KUKA KRL program: MyProgram_154().src

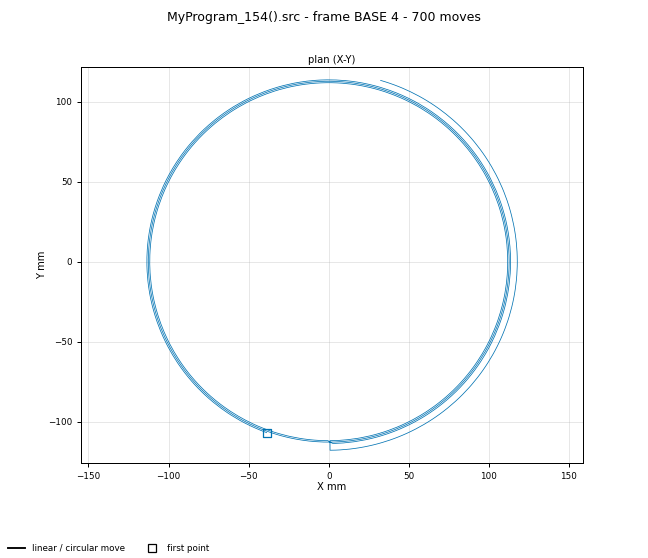
[picture p0: tool path of MyProgram_154().src in frame BASE 4, 700 of 700 moves have a stored position in this frame; points joined in program order, loops and branches not executed]
&ACCESS RVP
&REL 1
&PARAM TEMPLATE = C:\KRC\Roboter\Template\vorgabe
&PARAM EDITMASK = *
DEF MyProgram_154()
; ---- Setting reference (Base) ----
$BASE = BASE_DATA[4]

; --------------------------
; ---- Setting tool (TCP) ----
$TOOL = TOOL_DATA[3]
; --------------------------

$VEL.CP = VEL_APROX_PRINT
Startdeposition()
$VEL.CP = VEL_PRINT
LIN {X -38.7795,Y -106.7145,Z 119,A -114.0854,B 24.9553,C -1.5455,E1 24.9444,E2 200.0846} C_DIS
LIN {X -42.2899,Y -105.3741,Z 119,A -116.1743,B 24.9556,C -1.5393,E1 24.9389,E2 202.1927} C_DIS
LIN {X -46.3885,Y -103.634,Z 119,A -118.1057,B 24.9547,C -1.5549,E1 24.9341,E2 204.0916} C_DIS
LIN {X -48.9846,Y -102.4323,Z 119,A -120.2238,B 24.9562,C -1.5287,E1 24.9286,E2 206.2774} C_DIS
LIN {X -52.6968,Y -100.573,Z 119,A -121.7129,B 24.9546,C -1.5564,E1 24.925,E2 207.7047} C_DIS
LIN {X -55.5486,Y -99.0263,Z 119,A -123.3546,B 24.9545,C -1.5584,E1 24.921,E2 209.3463} C_DIS
LIN {X -60.9242,Y -95.8139,Z 119,A -126.6405,B 24.9545,C -1.5579,E1 24.9132,E2 212.6435} C_DIS
LIN {X -63.1418,Y -94.368,Z 119,A -128.2578,B 24.9551,C -1.5485,E1 24.9093,E2 214.2885} C_DIS
LIN {X -67.1706,Y -91.542,Z 119,A -130.4641,B 24.9542,C -1.5641,E1 24.9044,E2 216.4654} C_DIS
LIN {X -70.0841,Y -89.3319,Z 119,A -132.2235,B 24.9538,C -1.571,E1 24.9005,E2 218.2149} C_DIS
LIN {X -71.9862,Y -87.8078,Z 119,A -133.5514,B 24.9538,C -1.5692,E1 24.8976,E2 219.5519} C_DIS
LIN {X -74.7924,Y -85.428,Z 119,A -135.353,B 24.9535,C -1.5751,E1 24.8938,E2 221.3466} C_DIS
LIN {X -77.6668,Y -82.8234,Z 119,A -137.329,B 24.9533,C -1.5784,E1 24.8898,E2 223.3229} C_DIS
LIN {X -81.3821,Y -79.1774,Z 119,A -140.0426,B 24.9532,C -1.5804,E1 24.8844,E2 226.043} C_DIS
LIN {X -83.7193,Y -76.7001,Z 119,A -141.611,B 24.9526,C -1.5904,E1 24.8814,E2 227.5946} C_DIS
LIN {X -85.8302,Y -74.3318,Z 119,A -143.3683,B 24.9528,C -1.5877,E1 24.8782,E2 229.3661} C_DIS
LIN {X -88.2166,Y -71.4818,Z 119,A -145.143,B 24.9523,C -1.5962,E1 24.875,E2 231.1288} C_DIS
LIN {X -90.1414,Y -69.0395,Z 119,A -147.103,B 24.953,C -1.5844,E1 24.8716,E2 233.1262} C_DIS
LIN {X -92.0799,Y -66.4339,Z 119,A -148.4579,B 24.952,C -1.5998,E1 24.8694,E2 234.451} C_DIS
LIN {X -94.3065,Y -63.2327,Z 119,A -151.3484,B 24.9539,C -1.5684,E1 24.8648,E2 237.4308} C_DIS
LIN {X -97.447,Y -58.2773,Z 119,A -153.2453,B 24.9509,C -1.6182,E1 24.8622,E2 239.2187} C_DIS
LIN {X -100.3495,Y -53.1211,Z 119,A -156.2923,B 24.9506,C -1.6239,E1 24.8581,E2 242.2681} C_DIS
LIN {X -101.8163,Y -50.2524,Z 119,A -157.9977,B 24.9505,C -1.6253,E1 24.8559,E2 243.9793} C_DIS
LIN {X -103.469,Y -46.7547,Z 119,A -160.1125,B 24.9505,C -1.6245,E1 24.8534,E2 246.1077} C_DIS
LIN {X -105.0495,Y -43.0873,Z 119,A -161.9877,B 24.9499,C -1.6359,E1 24.8514,E2 247.9662} C_DIS
LIN {X -107.1276,Y -37.6231,Z 119,A -164.846,B 24.9491,C -1.6482,E1 24.8486,E2 250.811} C_DIS
LIN {X -108.4347,Y -33.6711,Z 119,A -167.0827,B 24.9491,C -1.6492,E1 24.8467,E2 253.0583} C_DIS
LIN {X -109.4832,Y -30.0915,Z 119,A -169.0013,B 24.9488,C -1.6535,E1 24.8452,E2 254.9776} C_DIS
LIN {X -110.3079,Y -26.9068,Z 119,A -170.6364,B 24.9484,C -1.6597,E1 24.8441,E2 256.6076} C_DIS
LIN {X -111.1636,Y -23.1205,Z 119,A -172.5881,B 24.948,C -1.6661,E1 24.8429,E2 258.5555} C_DIS
LIN {X -111.7921,Y -19.8596,Z 119,A -174.5884,B 24.9484,C -1.6587,E1 24.8419,E2 260.5853} C_DIS
LIN {X -112.5109,Y -15.2835,Z 119,A -176.6425,B 24.9473,C -1.6772,E1 24.8411,E2 262.6076} C_DIS
LIN {X -112.9126,Y -11.9401,Z 119,A -178.5887,B 24.9475,C -1.673,E1 24.8405,E2 264.5754} C_DIS
LIN {X -113.3804,Y -6.0614,Z 119,A 178.5739,B 24.9466,C -1.688,E1 24.84,E2 267.3941} C_DIS
LIN {X -113.5197,Y -2.2658,Z 119,A 176.7243,B 24.946,C -1.6968,E1 24.8398,E2 269.2338} C_DIS
LIN {X -113.5092,Y 2.8146,Z 119,A 173.8444,B 24.9463,C -1.6928,E1 24.8398,E2 272.1406} C_DIS
LIN {X -113.2912,Y 7.5449,Z 119,A 171.7176,B 24.9451,C -1.7109,E1 24.8402,E2 274.2372} C_DIS
LIN {X -113.0207,Y 10.8788,Z 119,A 170.163,B 24.9445,C -1.7216,E1 24.8406,E2 275.7756} C_DIS
LIN {X -112.6461,Y 14.2411,Z 119,A 168.2727,B 24.9445,C -1.72,E1 24.8412,E2 277.6811} C_DIS
LIN {X -112.0315,Y 18.4615,Z 119,A 166.1494,B 24.944,C -1.7281,E1 24.8421,E2 279.7977} C_DIS
LIN {X -111.4363,Y 21.7683,Z 119,A 164.3501,B 24.944,C -1.7295,E1 24.843,E2 281.6042} C_DIS
LIN {X -110.5057,Y 26.0885,Z 119,A 161.6768,B 24.9446,C -1.7195,E1 24.8447,E2 284.3172} C_DIS
LIN {X -109.5791,Y 29.7363,Z 119,A 160.2216,B 24.9431,C -1.7428,E1 24.8457,E2 285.7252} C_DIS
LIN {X -108.4418,Y 33.648,Z 119,A 157.5317,B 24.9443,C -1.7247,E1 24.848,E2 288.4737} C_DIS
LIN {X -106.9969,Y 37.9954,Z 119,A 155.7728,B 24.9424,C -1.7533,E1 24.8496,E2 290.1743} C_DIS
LIN {X -105.7047,Y 41.4529,Z 119,A 154.0435,B 24.9417,C -1.7644,E1 24.8513,E2 291.8871} C_DIS
LIN {X -103.2381,Y 47.267,Z 119,A 150.8158,B 24.9411,C -1.7725,E1 24.8548,E2 295.1133} C_DIS
LIN {X -101.4731,Y 50.9447,Z 119,A 148.6316,B 24.9411,C -1.7737,E1 24.8575,E2 297.3062} C_DIS
LIN {X -99.5576,Y 54.5927,Z 119,A 146.5283,B 24.9407,C -1.779,E1 24.8603,E2 299.4083} C_DIS
LIN {X -97.1628,Y 58.7474,Z 119,A 144.0709,B 24.9403,C -1.7845,E1 24.8638,E2 301.8651} C_DIS
LIN {X -95.0134,Y 62.1645,Z 119,A 142.116,B 24.9397,C -1.7935,E1 24.8667,E2 303.8084} C_DIS
LIN {X -91.9767,Y 66.5766,Z 119,A 139.0093,B 24.9403,C -1.7852,E1 24.8717,E2 306.9502} C_DIS
LIN {X -89.9849,Y 69.2426,Z 119,A 137.365,B 24.9399,C -1.7911,E1 24.8745,E2 308.5882} C_DIS
LIN {X -87.9451,Y 71.8168,Z 119,A 136.1646,B 24.9384,C -1.8135,E1 24.8766,E2 309.7409} C_DIS
LIN {X -85.2574,Y 74.9865,Z 119,A 133.7554,B 24.9388,C -1.8066,E1 24.881,E2 312.1775} C_DIS
LIN {X -80.3903,Y 80.1843,Z 119,A 130.2401,B 24.938,C -1.8186,E1 24.8878,E2 315.6795} C_DIS
LIN {X -77.9973,Y 82.5126,Z 119,A 128.0362,B 24.9391,C -1.8021,E1 24.8923,E2 317.9316} C_DIS
LIN {X -74.8259,Y 85.3987,Z 119,A 125.7336,B 24.9391,C -1.8016,E1 24.8972,E2 320.2445} C_DIS
LIN {X -71.0662,Y 88.5534,Z 119,A 123.8711,B 24.9371,C -1.8314,E1 24.9011,E2 322.0433} C_DIS
LIN {X -68.7439,Y 90.3689,Z 119,A 121.8998,B 24.9382,C -1.8153,E1 24.9056,E2 324.0599} C_DIS
LIN {X -65.3509,Y 92.8521,Z 119,A 120.2399,B 24.9367,C -1.838,E1 24.9092,E2 325.6716} C_DIS
LIN {X -61.8864,Y 95.1962,Z 119,A 118.1045,B 24.9365,C -1.8411,E1 24.9142,E2 327.8066} C_DIS
LIN {X -59.1389,Y 96.925,Z 119,A 115.4465,B 24.939,C -1.8036,E1 24.9208,E2 330.562} C_DIS
LIN {X -53.3558,Y 100.2259,Z 119,A 113.1232,B 24.9358,C -1.8507,E1 24.9262,E2 332.7797} C_DIS
LIN {X -50.2914,Y 101.7969,Z 119,A 111.6116,B 24.935,C -1.8628,E1 24.9299,E2 334.2669} C_DIS
LIN {X -46.3293,Y 103.6607,Z 119,A 109.3479,B 24.9349,C -1.8639,E1 24.9357,E2 336.5333} C_DIS
LIN {X -40.3596,Y 106.127,Z 119,A 105.8317,B 24.9353,C -1.858,E1 24.9448,E2 340.0714} C_DIS
LIN {X -36.0067,Y 107.682,Z 119,A 103.3217,B 24.9356,C -1.8537,E1 24.9515,E2 342.5964} C_DIS
LIN {X -31.3299,Y 109.1348,Z 119,A 101.1768,B 24.9345,C -1.8698,E1 24.9571,E2 344.7067} C_DIS
LIN {X -28.2896,Y 109.9614,Z 119,A 99.6621,B 24.9341,C -1.8745,E1 24.9612,E2 346.2124} C_DIS
LIN {X -22.2676,Y 111.3387,Z 119,A 96.426,B 24.9343,C -1.8724,E1 24.9701,E2 349.4577} C_DIS
LIN {X -18.8866,Y 111.9604,Z 119,A 94.8799,B 24.9336,C -1.8815,E1 24.9742,E2 350.9837} C_DIS
LIN {X -13.7991,Y 112.7021,Z 119,A 92.1188,B 24.934,C -1.8762,E1 24.9819,E2 353.7596} C_DIS
LIN {X -7.9378,Y 113.2647,Z 119,A 89.1949,B 24.9338,C -1.8797,E1 24.99,E2 356.6768} C_DIS
LIN {X -5.1434,Y 113.4259,Z 119,A 87.1623,B 24.9355,C -1.8543,E1 24.9959,E2 358.77} C_DIS
LIN {X -1.0062,Y 113.5381,Z 119,A 85.4495,B 24.9344,C -1.8704,E1 25.0006,E2 360.4446} C_DIS
LIN {X 4.6202,Y 113.4484,Z 119,A 82.9834,B 24.9333,C -1.8865,E1 25.0073,E2 362.8722} C_DIS
LIN {X 10.4517,Y 113.0601,Z 119,A 79.3073,B 24.9354,C -1.8557,E1 25.0178,E2 366.6194} C_DIS
LIN {X 14.4604,Y 112.6176,Z 119,A 77.7972,B 24.9339,C -1.8775,E1 25.0218,E2 368.0768} C_DIS
LIN {X 17.49,Y 112.1871,Z 119,A 75.8625,B 24.9351,C -1.8604,E1 25.0272,E2 370.0501} C_DIS
LIN {X 20.9601,Y 111.5919,Z 119,A 74.3788,B 24.9343,C -1.8721,E1 25.0312,E2 371.5044} C_DIS
LIN {X 25.1759,Y 110.7165,Z 119,A 72.3191,B 24.934,C -1.8759,E1 25.0368,E2 373.5525} C_DIS
LIN {X 28.519,Y 109.9025,Z 119,A 70.6003,B 24.934,C -1.8756,E1 25.0415,E2 375.2693} C_DIS
LIN {X 32.1679,Y 108.8901,Z 119,A 68.6954,B 24.9341,C -1.8745,E1 25.0466,E2 377.1736} C_DIS
LIN {X 35.545,Y 107.8367,Z 119,A 66.9758,B 24.9341,C -1.8759,E1 25.0511,E2 378.8868} C_DIS
LIN {X 37.8064,Y 107.0633,Z 119,A 65.6314,B 24.9345,C -1.8689,E1 25.0547,E2 380.2451} C_DIS
LIN {X 42.254,Y 105.3886,Z 119,A 63.2762,B 24.9345,C -1.8684,E1 25.0609,E2 382.5965} C_DIS
LIN {X 45.7399,Y 103.9223,Z 119,A 60.8053,B 24.9364,C -1.8419,E1 25.0673,E2 385.1239} C_DIS
LIN {X 49.6347,Y 102.1199,Z 119,A 59.1837,B 24.935,C -1.8628,E1 25.0713,E2 386.6919} C_DIS
LIN {X 53.4516,Y 100.1754,Z 119,A 56.6902,B 24.9362,C -1.8455,E1 25.0775,E2 389.2194} C_DIS
LIN {X 56.3394,Y 98.5787,Z 119,A 55.1408,B 24.936,C -1.8481,E1 25.0813,E2 390.7579} C_DIS
LIN {X 60.8663,Y 95.851,Z 119,A 52.6168,B 24.9358,C -1.8503,E1 25.0872,E2 393.2688} C_DIS
LIN {X 64.1193,Y 93.7061,Z 119,A 50.6128,B 24.9362,C -1.8454,E1 25.0919,E2 395.2776} C_DIS
LIN {X 67.6543,Y 91.1875,Z 119,A 48.5006,B 24.9362,C -1.845,E1 25.0966,E2 397.3834} C_DIS
LIN {X 71.9271,Y 87.8557,Z 119,A 45.7992,B 24.9364,C -1.8413,E1 25.1025,E2 400.0833} C_DIS
LIN {X 74.6558,Y 85.5473,Z 119,A 44.2974,B 24.9358,C -1.8512,E1 25.1057,E2 401.5558} C_DIS
LIN {X 78.3837,Y 82.1471,Z 119,A 41.4962,B 24.9369,C -1.8346,E1 25.1115,E2 404.3849} C_DIS
LIN {X 81.1101,Y 79.4556,Z 119,A 39.7544,B 24.9366,C -1.839,E1 25.1149,E2 406.109} C_DIS
LIN {X 84.2332,Y 76.1372,Z 119,A 37.2848,B 24.9375,C -1.8262,E1 25.1196,E2 408.598} C_DIS
LIN {X 86.7497,Y 73.2567,Z 119,A 34.8821,B 24.9392,C -1.8005,E1 25.124,E2 411.0503} C_DIS
LIN {X 89.3227,Y 70.0958,Z 119,A 33.3055,B 24.9381,C -1.817,E1 25.1267,E2 412.5805} C_DIS
LIN {X 91.5873,Y 67.1087,Z 119,A 31.7955,B 24.9373,C -1.8296,E1 25.1292,E2 414.0537} C_DIS
LIN {X 93.2489,Y 64.78,Z 119,A 30.0633,B 24.9384,C -1.8128,E1 25.132,E2 415.8169} C_DIS
LIN {X 94.9753,Y 62.2223,Z 119,A 28.4277,B 24.9389,C -1.8052,E1 25.1345,E2 417.4624} C_DIS
LIN {X 96.9762,Y 59.0546,Z 119,A 26.5962,B 24.9391,C -1.8029,E1 25.1372,E2 419.2901} C_DIS
LIN {X 98.9328,Y 55.7161,Z 119,A 24.6472,B 24.9394,C -1.7977,E1 25.1399,E2 421.2412} C_DIS
LIN {X 100.7803,Y 52.303,Z 119,A 22.8234,B 24.9394,C -1.7984,E1 25.1423,E2 423.0538} C_DIS
LIN {X 104.3637,Y 44.7269,Z 119,A 18.6192,B 24.9401,C -1.7874,E1 25.1473,E2 427.2613} C_DIS
LIN {X 106.2287,Y 40.0912,Z 119,A 16.0223,B 24.9408,C -1.7765,E1 25.15,E2 429.8695} C_DIS
LIN {X 107.5213,Y 36.4834,Z 119,A 14.1733,B 24.941,C -1.7746,E1 25.1517,E2 431.7127} C_DIS
LIN {X 108.4396,Y 33.6552,Z 119,A 12.6614,B 24.9413,C -1.7695,E1 25.1529,E2 433.228} C_DIS
LIN {X 109.6687,Y 29.4048,Z 119,A 10.3479,B 24.942,C -1.7589,E1 25.1547,E2 435.5532} C_DIS
LIN {X 110.5233,Y 26.0121,Z 119,A 8.1985,B 24.9435,C -1.7358,E1 25.1561,E2 437.7445} C_DIS
LIN {X 111.3121,Y 22.397,Z 119,A 6.9312,B 24.9421,C -1.7574,E1 25.1568,E2 438.9535} C_DIS
LIN {X 112.0752,Y 18.197,Z 119,A 4.421,B 24.9436,C -1.7342,E1 25.158,E2 441.5036} C_DIS
LIN {X 112.6423,Y 14.2702,Z 119,A 1.9254,B 24.9455,C -1.7053,E1 25.1589,E2 444.0527} C_DIS
LIN {X 113.1592,Y 9.3219,Z 119,A -0.513,B 24.9458,C -1.7005,E1 25.1595,E2 446.4881} C_DIS
LIN {X 113.4497,Y 4.59,Z 119,A -2.2614,B 24.9444,C -1.7222,E1 25.1597,E2 448.1749} C_DIS
LIN {X 113.5358,Y 1.3367,Z 119,A -3.9301,B 24.9448,C -1.7156,E1 25.1597,E2 449.8491} C_DIS
LIN {X 113.5269,Y -1.8736,Z 119,A -5.7164,B 24.9457,C -1.7027,E1 25.1597,E2 451.6552} C_DIS
LIN {X 113.3099,Y -7.2693,Z 119,A -7.9332,B 24.9447,C -1.7173,E1 25.1594,E2 453.8247} C_DIS
LIN {X 112.6463,Y -14.239,Z 119,A -11.8061,B 24.9465,C -1.69,E1 25.1583,E2 457.7389} C_DIS
LIN {X 111.7509,Y -20.0885,Z 119,A -14.4516,B 24.9461,C -1.696,E1 25.1572,E2 460.3546} C_DIS
LIN {X 110.4229,Y -26.4358,Z 119,A -17.8457,B 24.9471,C -1.6797,E1 25.1552,E2 463.7673} C_DIS
LIN {X 109.6822,Y -29.3549,Z 119,A -19.3799,B 24.9475,C -1.6742,E1 25.1541,E2 465.3058} C_DIS
LIN {X 108.6814,Y -32.8714,Z 119,A -21.317,B 24.9481,C -1.6641,E1 25.1525,E2 467.2557} C_DIS
LIN {X 107.5918,Y -36.2743,Z 119,A -22.9036,B 24.9478,C -1.6684,E1 25.1512,E2 468.8232} C_DIS
LIN {X 106.354,Y -39.7601,Z 119,A -24.9096,B 24.9486,C -1.6561,E1 25.1493,E2 470.8469} C_DIS
LIN {X 103.6092,Y -46.4435,Z 119,A -28.1919,B 24.9483,C -1.6616,E1 25.1458,E2 474.0982} C_DIS
LIN {X 101.598,Y -50.6927,Z 119,A -30.8862,B 24.9496,C -1.6395,E1 25.1425,E2 476.83} C_DIS
LIN {X 99.7763,Y -54.1897,Z 119,A -33.2879,B 24.9511,C -1.6147,E1 25.1392,E2 479.2775} C_DIS
LIN {X 97.8977,Y -57.5148,Z 119,A -34.6108,B 24.9498,C -1.6367,E1 25.1375,E2 480.5418} C_DIS
LIN {X 94.8546,Y -62.4054,Z 119,A -37.612,B 24.9506,C -1.624,E1 25.133,E2 483.5578} C_DIS
LIN {X 93.2011,Y -64.8488,Z 119,A -38.953,B 24.9504,C -1.6266,E1 25.1309,E2 484.8861} C_DIS
LIN {X 91.3605,Y -67.4186,Z 119,A -40.6904,B 24.9511,C -1.6156,E1 25.128,E2 486.641} C_DIS
LIN {X 89.2292,Y -70.2141,Z 119,A -42.384,B 24.9511,C -1.6145,E1 25.1251,E2 488.3292} C_DIS
LIN {X 87.0673,Y -72.8784,Z 119,A -44.2734,B 24.9519,C -1.6027,E1 25.1217,E2 490.2378} C_DIS
LIN {X 84.57,Y -75.7611,Z 119,A -46.063,B 24.9519,C -1.6038,E1 25.1184,E2 492.0166} C_DIS
LIN {X 81.984,Y -78.5529,Z 119,A -48.0162,B 24.9522,C -1.5975,E1 25.1147,E2 493.9763} C_DIS
LIN {X 79.4027,Y -81.1624,Z 119,A -49.9139,B 24.9526,C -1.5908,E1 25.1109,E2 495.8816} C_DIS
LIN {X 76.7767,Y -83.649,Z 119,A -51.633,B 24.9526,C -1.5913,E1 25.1074,E2 497.5926} C_DIS
LIN {X 73.944,Y -86.1642,Z 119,A -53.5598,B 24.9529,C -1.5862,E1 25.1034,E2 499.5239} C_DIS
LIN {X 71.6521,Y -88.0786,Z 119,A -55.058,B 24.953,C -1.5832,E1 25.1001,E2 501.0235} C_DIS
LIN {X 68.6736,Y -90.4218,Z 119,A -57.0278,B 24.9534,C -1.5764,E1 25.0958,E2 503.002} C_DIS
LIN {X 66.0008,Y -92.3889,Z 119,A -58.6322,B 24.9534,C -1.5761,E1 25.0921,E2 504.6015} C_DIS
LIN {X 62.724,Y -94.6446,Z 119,A -60.4684,B 24.9532,C -1.5798,E1 25.0879,E2 506.4229} C_DIS
LIN {X 60.2833,Y -96.2173,Z 119,A -62.0206,B 24.9536,C -1.573,E1 25.0843,E2 507.9861} C_DIS
LIN {X 57.7569,Y -97.7546,Z 119,A -63.5157,B 24.9538,C -1.5701,E1 25.0807,E2 509.4834} C_DIS
LIN {X 53.4628,Y -100.1696,Z 119,A -66.1549,B 24.9545,C -1.5588,E1 25.0742,E2 512.1417} C_DIS
LIN {X 50.0811,Y -101.9012,Z 119,A -67.9524,B 24.9543,C -1.5609,E1 25.0697,E2 513.9291} C_DIS
LIN {X 44.5083,Y -104.4551,Z 119,A -71.2636,B 24.9552,C -1.5465,E1 25.0612,E2 517.2663} C_DIS
LIN {X 40.6633,Y -106.012,Z 119,A -73.3415,B 24.9553,C -1.5442,E1 25.0558,E2 519.345} C_DIS
LIN {X 36.415,Y -107.5443,Z 119,A -75.407,B 24.9549,C -1.5507,E1 25.0504,E2 521.3909} C_DIS
LIN {X 33.2505,Y -108.5651,Z 119,A -77.1473,B 24.9552,C -1.546,E1 25.0458,E2 523.1393} C_DIS
LIN {X 30.1039,Y -109.4798,Z 119,A -78.6676,B 24.955,C -1.55,E1 25.0417,E2 524.6476} C_DIS
LIN {X 26.8253,Y -110.3278,Z 119,A -80.324,B 24.955,C -1.5506,E1 25.0372,E2 526.3002} C_DIS
LIN {X 22.8635,Y -111.2164,Z 119,A -82.5574,B 24.9555,C -1.5406,E1 25.0311,E2 528.5543} C_DIS
LIN {X 15.9868,Y -112.411,Z 119,A -86.1378,B 24.9558,C -1.5354,E1 25.0212,E2 532.1434} C_DIS
LIN {X 9.0633,Y -113.1798,Z 119,A -90.5647,B 24.9582,C -1.4943,E1 25.0086,E2 536.6649} C_DIS
LIN {X 2.6596,Y -113.5124,Z 119,A -93.7317,B 24.9581,C -1.4962,E1 24.9998,E2 539.8268} C_DIS
LIN {X 2.6596,Y -113.5124,Z 119,A -93.7317,B 24.9581,C -1.4962,E1 24.9998,E2 539.8268} C_DIS
Enddeposition()
LIN {X 0.7947,Y -112.634,Z 119,A -93.4663,B 24.9542,C -1.5636,E1 25.001,E2 539.4018} C_DIS
Startdeposition()
$VEL.CP = VEL_PRINT
LIN {X 3.6315,Y -112.5922,Z 119,A -91.4349,B 24.9527,C -1.5892,E1 25.0068,E2 537.3099} C_DIS
LIN {X 9.3853,Y -112.2597,Z 119,A -88.603,B 24.9529,C -1.5862,E1 25.0147,E2 534.4866} C_DIS
LIN {X 14.6247,Y -111.6973,Z 119,A -85.9699,B 24.9529,C -1.5857,E1 25.022,E2 531.8565} C_DIS
LIN {X 17.4837,Y -111.2859,Z 119,A -84.4862,B 24.9528,C -1.5874,E1 25.0261,E2 530.3701} C_DIS
LIN {X 20.076,Y -110.8473,Z 119,A -82.5788,B 24.9512,C -1.6137,E1 25.0315,E2 528.4026} C_DIS
LIN {X 23.8423,Y -110.0987,Z 119,A -81.0612,B 24.9523,C -1.5961,E1 25.0355,E2 526.9285} C_DIS
LIN {X 27.3941,Y -109.271,Z 119,A -79.1677,B 24.9521,C -1.5996,E1 25.0407,E2 525.0295} C_DIS
LIN {X 31.0805,Y -108.2788,Z 119,A -77.4071,B 24.9524,C -1.5937,E1 25.0454,E2 523.2856} C_DIS
LIN {X 34.4302,Y -107.2604,Z 119,A -75.5291,B 24.952,C -1.6002,E1 25.0504,E2 521.3958} C_DIS
LIN {X 37.9515,Y -106.0675,Z 119,A -73.1772,B 24.9506,C -1.6232,E1 25.0567,E2 518.9941} C_DIS
LIN {X 41.4531,Y -104.7467,Z 119,A -71.8213,B 24.9519,C -1.6014,E1 25.0601,E2 517.6929} C_DIS
LIN {X 47.4616,Y -102.1644,Z 119,A -68.809,B 24.9525,C -1.5923,E1 25.0678,E2 514.7093} C_DIS
LIN {X 50.1295,Y -100.8821,Z 119,A -66.9839,B 24.9515,C -1.6091,E1 25.0724,E2 512.8494} C_DIS
LIN {X 53.2616,Y -99.2654,Z 119,A -65.1317,B 24.9511,C -1.6148,E1 25.077,E2 510.9888} C_DIS
LIN {X 57.1934,Y -97.052,Z 119,A -62.9315,B 24.9511,C -1.6148,E1 25.0823,E2 508.7954} C_DIS
LIN {X 59.8016,Y -95.467,Z 119,A -61.1759,B 24.9504,C -1.6269,E1 25.0866,E2 507.0167} C_DIS
LIN {X 63.4757,Y -93.0652,Z 119,A -59.1345,B 24.9507,C -1.6227,E1 25.0913,E2 504.992} C_DIS
LIN {X 66.5163,Y -90.9161,Z 119,A -57.2466,B 24.9504,C -1.6264,E1 25.0955,E2 503.102} C_DIS
LIN {X 69.2022,Y -88.8905,Z 119,A -55.4209,B 24.9499,C -1.6353,E1 25.0996,E2 501.262} C_DIS
LIN {X 72.0223,Y -86.6195,Z 119,A -53.6859,B 24.9499,C -1.6346,E1 25.1033,E2 499.5353} C_DIS
LIN {X 74.8907,Y -84.1526,Z 119,A -51.7388,B 24.9496,C -1.6401,E1 25.1074,E2 497.583} C_DIS
LIN {X 77.4696,Y -81.7849,Z 119,A -49.9042,B 24.9492,C -1.6468,E1 25.1112,E2 495.7399} C_DIS
LIN {X 80.1076,Y -79.2019,Z 119,A -48.1676,B 24.9492,C -1.6449,E1 25.1146,E2 494.0151} C_DIS
LIN {X 82.5016,Y -76.7076,Z 119,A -46.3106,B 24.9487,C -1.6539,E1 25.1182,E2 492.145} C_DIS
LIN {X 84.8864,Y -74.0571,Z 119,A -44.5965,B 24.9487,C -1.654,E1 25.1214,E2 490.4382} C_DIS
LIN {X 87.368,Y -71.1129,Z 119,A -42.6253,B 24.9484,C -1.6598,E1 25.1249,E2 488.4624} C_DIS
LIN {X 89.4115,Y -68.5261,Z 119,A -41.0209,B 24.9483,C -1.661,E1 25.1276,E2 486.8628} C_DIS
LIN {X 91.5304,Y -65.6691,Z 119,A -38.8766,B 24.947,C -1.6815,E1 25.1312,E2 484.6805} C_DIS
LIN {X 93.5113,Y -62.8169,Z 119,A -37.2723,B 24.9472,C -1.679,E1 25.1337,E2 483.0901} C_DIS
LIN {X 97.5682,Y -56.3084,Z 119,A -33.5204,B 24.9469,C -1.6833,E1 25.1391,E2 479.347} C_DIS
LIN {X 99.4537,Y -52.9087,Z 119,A -31.5202,B 24.9465,C -1.6903,E1 25.1418,E2 477.3409} C_DIS
LIN {X 101.2342,Y -49.4193,Z 119,A -29.415,B 24.9457,C -1.7015,E1 25.1444,E2 475.2206} C_DIS
LIN {X 102.9456,Y -45.7461,Z 119,A -27.4796,B 24.9457,C -1.702,E1 25.1467,E2 473.2946} C_DIS
LIN {X 105.0232,Y -40.7492,Z 119,A -24.6819,B 24.945,C -1.7126,E1 25.1496,E2 470.4872} C_DIS
LIN {X 106.3578,Y -37.1242,Z 119,A -22.9296,B 24.9453,C -1.7089,E1 25.1512,E2 468.7534} C_DIS
LIN {X 107.4241,Y -33.9199,Z 119,A -21.0792,B 24.9445,C -1.7205,E1 25.1528,E2 466.8862} C_DIS
LIN {X 108.4494,Y -30.4786,Z 119,A -19.2611,B 24.9442,C -1.726,E1 25.1543,E2 465.0656} C_DIS
LIN {X 109.5508,Y -26.2486,Z 119,A -17.2319,B 24.9442,C -1.7241,E1 25.1556,E2 463.0526} C_DIS
LIN {X 110.4204,Y -22.3072,Z 119,A -15.1724,B 24.9438,C -1.731,E1 25.1568,E2 460.9887} C_DIS
LIN {X 111.0009,Y -19.2193,Z 119,A -13.4091,B 24.943,C -1.7439,E1 25.1577,E2 459.2055} C_DIS
LIN {X 111.7852,Y -13.9466,Z 119,A -10.8296,B 24.9428,C -1.7466,E1 25.1587,E2 456.6347} C_DIS
LIN {X 112.3337,Y -8.4596,Z 119,A -8.174,B 24.9427,C -1.7488,E1 25.1594,E2 453.9897} C_DIS
LIN {X 112.5698,Y -4.2983,Z 119,A -5.6678,B 24.941,C -1.7736,E1 25.1597,E2 451.4398} C_DIS
LIN {X 112.6514,Y -0.0991,Z 119,A -3.5805,B 24.9407,C -1.7783,E1 25.1597,E2 449.3538} C_DIS
LIN {X 112.5859,Y 3.8355,Z 119,A -0.8985,B 24.9381,C -1.8167,E1 25.1595,E2 446.5974} C_DIS
LIN {X 112.2447,Y 9.5723,Z 119,A 1.1622,B 24.9402,C -1.7857,E1 25.1591,E2 444.6219} C_DIS
LIN {X 111.6524,Y 14.9717,Z 119,A 3.7608,B 24.9402,C -1.787,E1 25.1582,E2 442.0357} C_DIS
LIN {X 110.6446,Y 21.1646,Z 119,A 6.6735,B 24.9403,C -1.7842,E1 25.1569,E2 439.1465} C_DIS
LIN {X 109.7837,Y 25.2527,Z 119,A 9.1378,B 24.9388,C -1.8065,E1 25.1554,E2 436.6439} C_DIS
LIN {X 108.999,Y 28.4524,Z 119,A 10.6712,B 24.9389,C -1.8052,E1 25.1544,E2 435.1227} C_DIS
LIN {X 108.1951,Y 31.376,Z 119,A 12.3655,B 24.9381,C -1.8169,E1 25.1531,E2 433.4104} C_DIS
LIN {X 107.1483,Y 34.7766,Z 119,A 14.1339,B 24.9379,C -1.8205,E1 25.1516,E2 431.6435} C_DIS
LIN {X 105.8415,Y 38.5711,Z 119,A 16.1402,B 24.9376,C -1.825,E1 25.1497,E2 429.6378} C_DIS
LIN {X 104.2185,Y 42.764,Z 119,A 18.34,B 24.9374,C -1.8278,E1 25.1475,E2 427.4437} C_DIS
LIN {X 103.0183,Y 45.5824,Z 119,A 20.0598,B 24.9366,C -1.8397,E1 25.1455,E2 425.7052} C_DIS
LIN {X 100.3962,Y 51.0959,Z 119,A 22.739,B 24.9373,C -1.829,E1 25.1424,E2 423.0656} C_DIS
LIN {X 98.553,Y 54.5676,Z 119,A 25.0731,B 24.9359,C -1.8498,E1 25.1392,E2 420.6946} C_DIS
LIN {X 96.685,Y 57.8143,Z 119,A 26.852,B 24.9359,C -1.8492,E1 25.1367,E2 418.9263} C_DIS
LIN {X 94.8595,Y 60.7605,Z 119,A 28.6349,B 24.9355,C -1.8548,E1 25.134,E2 417.1393} C_DIS
LIN {X 93.0192,Y 63.5437,Z 119,A 30.2592,B 24.9355,C -1.8559,E1 25.1315,E2 415.5205} C_DIS
LIN {X 91.6445,Y 65.5092,Z 119,A 31.5461,B 24.935,C -1.862,E1 25.1294,E2 414.2254} C_DIS
LIN {X 89.559,Y 68.3347,Z 119,A 33.4497,B 24.9343,C -1.8718,E1 25.1262,E2 412.3078} C_DIS
LIN {X 86.938,Y 71.639,Z 119,A 35.5237,B 24.9342,C -1.8737,E1 25.1226,E2 410.239} C_DIS
LIN {X 84.814,Y 74.14,Z 119,A 37.1383,B 24.9341,C -1.8751,E1 25.1196,E2 408.6282} C_DIS
LIN {X 82.4097,Y 76.8052,Z 119,A 39.1339,B 24.9333,C -1.8869,E1 25.1158,E2 406.6136} C_DIS
LIN {X 79.115,Y 80.1933,Z 119,A 41.359,B 24.9335,C -1.8841,E1 25.1115,E2 404.4046} C_DIS
LIN {X 75.6509,Y 83.4719,Z 119,A 43.8839,B 24.9328,C -1.8935,E1 25.1063,E2 401.8678} C_DIS
LIN {X 72.9859,Y 85.8092,Z 119,A 45.5649,B 24.9329,C -1.8916,E1 25.1028,E2 400.1978} C_DIS
LIN {X 70.1723,Y 88.1258,Z 119,A 47.5785,B 24.9322,C -1.9023,E1 25.0984,E2 398.1667} C_DIS
LIN {X 66.7518,Y 90.7437,Z 119,A 49.5934,B 24.9324,C -1.8984,E1 25.0939,E2 396.1683} C_DIS
LIN {X 63.6728,Y 92.9318,Z 119,A 51.4063,B 24.9326,C -1.8968,E1 25.0898,E2 394.3653} C_DIS
LIN {X 61.1664,Y 94.599,Z 119,A 53.1385,B 24.9317,C -1.9082,E1 25.0857,E2 392.6119} C_DIS
LIN {X 58.6522,Y 96.1774,Z 119,A 55.7458,B 24.928,C -1.9595,E1 25.0792,E2 389.8912} C_DIS
LIN {X 52.6274,Y 99.6019,Z 119,A 57.8893,B 24.9321,C -1.9029,E1 25.0743,E2 387.8879} C_DIS
LIN {X 50.0218,Y 100.9355,Z 119,A 59.5599,B 24.9314,C -1.9128,E1 25.07,E2 386.1984} C_DIS
LIN {X 46.1351,Y 102.7703,Z 119,A 61.6921,B 24.9314,C -1.913,E1 25.0646,E2 384.0712} C_DIS
LIN {X 43.4758,Y 103.9235,Z 119,A 63.3061,B 24.9308,C -1.9207,E1 25.0605,E2 382.4427} C_DIS
LIN {X 39.2626,Y 105.5891,Z 119,A 65.4173,B 24.9313,C -1.9145,E1 25.055,E2 380.3507} C_DIS
LIN {X 35.7967,Y 106.8119,Z 119,A 66.9886,B 24.9321,C -1.9033,E1 25.051,E2 378.8093} C_DIS
LIN {X 33.5511,Y 107.5384,Z 119,A 68.5603,B 24.9309,C -1.9203,E1 25.0467,E2 377.2002} C_DIS
LIN {X 30.061,Y 108.5677,Z 119,A 70.3307,B 24.931,C -1.9181,E1 25.0419,E2 375.438} C_DIS
LIN {X 27.8574,Y 109.152,Z 119,A 71.5005,B 24.931,C -1.9193,E1 25.0388,E2 374.2671} C_DIS
LIN {X 24.4877,Y 109.9579,Z 119,A 73.3366,B 24.9306,C -1.9234,E1 25.0337,E2 372.4238} C_DIS
LIN {X 21.3615,Y 110.6067,Z 119,A 74.863,B 24.9309,C -1.92,E1 25.0296,E2 370.9074} C_DIS
LIN {X 18.29,Y 111.1563,Z 119,A 76.4751,B 24.9308,C -1.9216,E1 25.0252,E2 369.2931} C_DIS
LIN {X 15.6813,Y 111.5539,Z 119,A 77.8491,B 24.9306,C -1.9233,E1 25.0213,E2 367.9163} C_DIS
LIN {X 12.539,Y 111.952,Z 119,A 79.5061,B 24.9305,C -1.9256,E1 25.0167,E2 366.2551} C_DIS
LIN {X 8.6877,Y 112.3155,Z 119,A 81.624,B 24.93,C -1.9322,E1 25.0108,E2 364.1228} C_DIS
LIN {X 4.7207,Y 112.5517,Z 119,A 83.5167,B 24.9304,C -1.9266,E1 25.0056,E2 362.2439} C_DIS
LIN {X 0.6724,Y 112.6486,Z 119,A 85.8653,B 24.9295,C -1.9386,E1 24.9989,E2 359.8671} C_DIS
LIN {X -2.5326,Y 112.623,Z 119,A 87.2746,B 24.9303,C -1.9288,E1 24.9951,E2 358.481} C_DIS
LIN {X -5.8185,Y 112.5009,Z 119,A 88.9345,B 24.9303,C -1.9277,E1 24.9904,E2 356.8234} C_DIS
LIN {X -9.8873,Y 112.2168,Z 119,A 91.0695,B 24.9303,C -1.9293,E1 24.9845,E2 354.6836} C_DIS
LIN {X -13.2277,Y 111.8713,Z 119,A 92.6185,B 24.9308,C -1.9217,E1 24.9802,E2 353.1517} C_DIS
LIN {X -17.2817,Y 111.3171,Z 119,A 94.3792,B 24.9318,C -1.9069,E1 24.9755,E2 351.4246} C_DIS
LIN {X -19.4135,Y 110.9664,Z 119,A 95.9601,B 24.9304,C -1.9262,E1 24.971,E2 349.7965} C_DIS
LIN {X -22.8708,Y 110.3047,Z 119,A 97.5601,B 24.9311,C -1.9168,E1 24.9667,E2 348.2169} C_DIS
LIN {X -27.0893,Y 109.3457,Z 119,A 99.7345,B 24.9313,C -1.9136,E1 24.9608,E2 346.0471} C_DIS
LIN {X -30.2716,Y 108.508,Z 119,A 101.5936,B 24.9309,C -1.9196,E1 24.9557,E2 344.171} C_DIS
LIN {X -34.149,Y 107.351,Z 119,A 103.9729,B 24.9301,C -1.9305,E1 24.9493,E2 341.7615} C_DIS
LIN {X -37.4393,Y 106.2472,Z 119,A 105.2703,B 24.9317,C -1.909,E1 24.946,E2 340.5128} C_DIS
LIN {X -40.2691,Y 105.2079,Z 119,A 107.7177,B 24.9291,C -1.9447,E1 24.9394,E2 337.9753} C_DIS
LIN {X -45.2689,Y 103.155,Z 119,A 109.6447,B 24.9318,C -1.9067,E1 24.9347,E2 336.1342} C_DIS
LIN {X -48.7254,Y 101.5677,Z 119,A 111.5159,B 24.9322,C -1.9011,E1 24.9299,E2 334.2715} C_DIS
LIN {X -51.7702,Y 100.0516,Z 119,A 113.3893,B 24.932,C -1.9041,E1 24.9252,E2 332.386} C_DIS
LIN {X -56.7579,Y 97.3094,Z 119,A 116.1061,B 24.9329,C -1.8917,E1 24.9187,E2 329.6907} C_DIS
LIN {X -59.9092,Y 95.3997,Z 119,A 118.0575,B 24.9329,C -1.8914,E1 24.914,E2 327.7341} C_DIS
LIN {X -63.2264,Y 93.234,Z 119,A 120.1046,B 24.9331,C -1.8887,E1 24.9093,E2 325.6865} C_DIS
LIN {X -66.4102,Y 90.9938,Z 119,A 122.39,B 24.9325,C -1.897,E1 24.904,E2 323.3735} C_DIS
LIN {X -69.7329,Y 88.4731,Z 119,A 124.6587,B 24.9325,C -1.8984,E1 24.899,E2 321.0931} C_DIS
LIN {X -72.4847,Y 86.2324,Z 119,A 126.2201,B 24.9334,C -1.8845,E1 24.8957,E2 319.5588} C_DIS
LIN {X -76.1549,Y 83.0095,Z 119,A 128.8601,B 24.9334,C -1.885,E1 24.8902,E2 316.907} C_DIS
LIN {X -79.2536,Y 80.0564,Z 119,A 131.6627,B 24.932,C -1.905,E1 24.8846,E2 314.045} C_DIS
LIN {X -83.2506,Y 75.8922,Z 119,A 133.8808,B 24.9345,C -1.8686,E1 24.8805,E2 311.9037} C_DIS
LIN {X -86.6876,Y 71.9404,Z 119,A 136.2597,B 24.9358,C -1.8504,E1 24.8762,E2 309.5576} C_DIS
LIN {X -88.6176,Y 69.5501,Z 119,A 138.7621,B 24.9335,C -1.8837,E1 24.8718,E2 306.9638} C_DIS
LIN {X -91.779,Y 65.3207,Z 119,A 140.62,B 24.9363,C -1.8432,E1 24.8689,E2 305.1934} C_DIS
LIN {X -93.2639,Y 63.1822,Z 119,A 141.9935,B 24.9364,C -1.8415,E1 24.8667,E2 303.8172} C_DIS
LIN {X -95.4963,Y 59.7547,Z 119,A 144.0525,B 24.9369,C -1.8347,E1 24.8636,E2 301.7639} C_DIS
LIN {X -97.6107,Y 56.2345,Z 119,A 146.8566,B 24.9354,C -1.8571,E1 24.8596,E2 298.8919} C_DIS
LIN {X -99.9054,Y 52.051,Z 119,A 148.5338,B 24.9379,C -1.8201,E1 24.8575,E2 297.294} C_DIS
LIN {X -101.5371,Y 48.7891,Z 119,A 150.4776,B 24.938,C -1.818,E1 24.8551,E2 295.3447} C_DIS
LIN {X -103.3382,Y 44.8486,Z 119,A 152.6665,B 24.9385,C -1.8107,E1 24.8526,E2 293.1612} C_DIS
LIN {X -104.8606,Y 41.1633,Z 119,A 154.7017,B 24.9389,C -1.8048,E1 24.8505,E2 291.1289} C_DIS
LIN {X -106.1927,Y 37.5948,Z 119,A 156.778,B 24.9389,C -1.8042,E1 24.8485,E2 289.0422} C_DIS
LIN {X -107.7489,Y 32.8724,Z 119,A 159.3249,B 24.9395,C -1.7969,E1 24.8463,E2 286.4981} C_DIS
LIN {X -108.7761,Y 29.2905,Z 119,A 161.1838,B 24.94,C -1.7894,E1 24.845,E2 284.6462} C_DIS
LIN {X -109.5649,Y 26.1908,Z 119,A 162.8452,B 24.9402,C -1.7856,E1 24.8439,E2 282.9843} C_DIS
LIN {X -110.2992,Y 22.8976,Z 119,A 164.5513,B 24.9406,C -1.7796,E1 24.8429,E2 281.2822} C_DIS
LIN {X -110.9418,Y 19.5504,Z 119,A 166.2997,B 24.941,C -1.7746,E1 24.842,E2 279.5355} C_DIS
LIN {X -111.4852,Y 16.165,Z 119,A 167.8086,B 24.942,C -1.7598,E1 24.8414,E2 278.053} C_DIS
LIN {X -111.7832,Y 13.9619,Z 119,A 169.0572,B 24.9419,C -1.7607,E1 24.8409,E2 276.7948} C_DIS
LIN {X -112.0526,Y 11.5929,Z 119,A 170.3541,B 24.9419,C -1.7601,E1 24.8405,E2 275.4915} C_DIS
LIN {X -112.3463,Y 8.3024,Z 119,A 172.1499,B 24.942,C -1.7591,E1 24.8401,E2 273.6873} C_DIS
LIN {X -112.5521,Y 4.7119,Z 119,A 173.8932,B 24.9426,C -1.7498,E1 24.8399,E2 271.9557} C_DIS
LIN {X -112.6444,Y 1.3551,Z 119,A 175.7384,B 24.9426,C -1.7496,E1 24.8398,E2 270.0998} C_DIS
LIN {X -112.6188,Y -2.7636,Z 119,A 177.7952,B 24.9432,C -1.7413,E1 24.8398,E2 268.0503} C_DIS
LIN {X -112.4574,Y -6.6052,Z 119,A 179.5646,B 24.9441,C -1.7277,E1 24.8401,E2 266.3028} C_DIS
LIN {X -112.2401,Y -9.6269,Z 119,A -178.841,B 24.9442,C -1.7248,E1 24.8405,E2 264.7057} C_DIS
LIN {X -111.9575,Y -12.4922,Z 119,A -177.3715,B 24.9445,C -1.7203,E1 24.8409,E2 263.2381} C_DIS
LIN {X -111.5173,Y -15.9393,Z 119,A -175.445,B 24.9445,C -1.721,E1 24.8416,E2 261.2986} C_DIS
LIN {X -110.9805,Y -19.3356,Z 119,A -173.8519,B 24.9452,C -1.7093,E1 24.8423,E2 259.7239} C_DIS
LIN {X -110.4669,Y -22.0809,Z 119,A -172.1982,B 24.9449,C -1.714,E1 24.8432,E2 258.0491} C_DIS
LIN {X -109.6155,Y -25.9811,Z 119,A -170.3333,B 24.9458,C -1.7011,E1 24.8444,E2 256.204} C_DIS
LIN {X -108.7764,Y -29.2892,Z 119,A -168.5543,B 24.946,C -1.6975,E1 24.8456,E2 254.4233} C_DIS
LIN {X -107.8023,Y -32.7001,Z 119,A -166.4608,B 24.9456,C -1.7034,E1 24.8473,E2 252.3035} C_DIS
LIN {X -106.5438,Y -36.5921,Z 119,A -164.5851,B 24.9465,C -1.689,E1 24.849,E2 250.4514} C_DIS
LIN {X -104.9578,Y -40.9156,Z 119,A -162.3281,B 24.9472,C -1.6787,E1 24.8512,E2 248.2063} C_DIS
LIN {X -103.7339,Y -43.9256,Z 119,A -160.5009,B 24.9471,C -1.6808,E1 24.8531,E2 246.3639} C_DIS
LIN {X -102.172,Y -47.4452,Z 119,A -158.6464,B 24.9477,C -1.6711,E1 24.8553,E2 244.5225} C_DIS
LIN {X -100.7425,Y -50.411,Z 119,A -156.9907,B 24.948,C -1.6656,E1 24.8573,E2 242.871} C_DIS
LIN {X -99.4866,Y -52.8463,Z 119,A -155.2553,B 24.9474,C -1.6754,E1 24.8596,E2 241.1029} C_DIS
LIN {X -96.9948,Y -57.2901,Z 119,A -152.9209,B 24.9485,C -1.6581,E1 24.8628,E2 238.7976} C_DIS
LIN {X -94.9948,Y -60.5497,Z 119,A -150.6118,B 24.9479,C -1.6676,E1 24.8663,E2 236.4542} C_DIS
LIN {X -92.3744,Y -64.4761,Z 119,A -148.5759,B 24.9492,C -1.6467,E1 24.8694,E2 234.4579} C_DIS
LIN {X -90.3518,Y -67.2825,Z 119,A -146.9607,B 24.9498,C -1.6365,E1 24.8721,E2 232.8592} C_DIS
LIN {X -88.72,Y -69.4205,Z 119,A -145.3534,B 24.9494,C -1.6428,E1 24.8749,E2 231.2291} C_DIS
LIN {X -86.5606,Y -72.0932,Z 119,A -143.6114,B 24.9497,C -1.6385,E1 24.8779,E2 229.4895} C_DIS
LIN {X -84.0625,Y -74.9913,Z 119,A -141.7081,B 24.9501,C -1.6323,E1 24.8814,E2 227.5923} C_DIS
LIN {X -82.1254,Y -77.1076,Z 119,A -140.2285,B 24.9502,C -1.6298,E1 24.8842,E2 226.112} C_DIS
LIN {X -79.4861,Y -79.8268,Z 119,A -138.2981,B 24.9505,C -1.6258,E1 24.888,E2 224.183} C_DIS
LIN {X -77.1762,Y -82.0609,Z 119,A -136.677,B 24.9507,C -1.6219,E1 24.8913,E2 222.5646} C_DIS
LIN {X -74.7599,Y -84.2696,Z 119,A -134.9575,B 24.9507,C -1.6207,E1 24.8949,E2 220.8409} C_DIS
LIN {X -71.8785,Y -86.739,Z 119,A -133.1099,B 24.9512,C -1.6137,E1 24.8988,E2 219.003} C_DIS
LIN {X -69.252,Y -88.8521,Z 119,A -131.242,B 24.951,C -1.6168,E1 24.9029,E2 217.1208} C_DIS
LIN {X -66.4872,Y -90.9374,Z 119,A -129.5602,B 24.9514,C -1.6104,E1 24.9067,E2 215.4481} C_DIS
LIN {X -62.5397,Y -93.6982,Z 119,A -126.9711,B 24.9514,C -1.6121,E1 24.9127,E2 212.8463} C_DIS
LIN {X -59.6112,Y -95.5859,Z 119,A -124.734,B 24.9503,C -1.6288,E1 24.9181,E2 210.5624} C_DIS
LIN {X -55.9905,Y -97.7509,Z 119,A -123.2723,B 24.9522,C -1.5972,E1 24.9214,E2 209.1716} C_DIS
LIN {X -53.4866,Y -99.1433,Z 119,A -121.67,B 24.952,C -1.6012,E1 24.9254,E2 207.5551} C_DIS
LIN {X -49.443,Y -101.2224,Z 119,A -119.4712,B 24.9524,C -1.5935,E1 24.9308,E2 205.3687} C_DIS
LIN {X -46.0541,Y -102.8068,Z 119,A -117.4324,B 24.9522,C -1.5971,E1 24.9361,E2 203.3165} C_DIS
LIN {X -42.7475,Y -104.2252,Z 119,A -115.6725,B 24.9525,C -1.5922,E1 24.9406,E2 201.5641} C_DIS
LIN {X -38.1197,Y -106.0061,Z 119,A -113.2268,B 24.9528,C -1.5866,E1 24.9469,E2 199.1266} C_DIS
LIN {X -35.5181,Y -106.9059,Z 119,A -111.6052,B 24.9523,C -1.5948,E1 24.9513,E2 197.4824} C_DIS
LIN {X -32.0125,Y -108.0063,Z 119,A -109.8897,B 24.9528,C -1.587,E1 24.9558,E2 195.7826} C_DIS
LIN {X -29.1796,Y -108.806,Z 119,A -108.4063,B 24.9529,C -1.5854,E1 24.9598,E2 194.3006} C_DIS
LIN {X -25.9214,Y -109.6292,Z 119,A -106.7534,B 24.9531,C -1.5821,E1 24.9643,E2 192.6534} C_DIS
LIN {X -22.8984,Y -110.299,Z 119,A -104.9893,B 24.9527,C -1.5894,E1 24.9692,E2 190.8696} C_DIS
LIN {X -19.9769,Y -110.8651,Z 119,A -103.5251,B 24.9528,C -1.5868,E1 24.9732,E2 189.4102} C_DIS
LIN {X -16.5445,Y -111.4311,Z 119,A -101.7311,B 24.9528,C -1.5873,E1 24.9781,E2 187.6133} C_DIS
LIN {X -12.2662,Y -111.982,Z 119,A -99.0779,B 24.9516,C -1.6069,E1 24.9856,E2 184.912} C_DIS
LIN {X -8.4322,Y -112.3359,Z 119,A -97.5262,B 24.9527,C -1.5892,E1 24.9898,E2 183.4016} C_DIS
LIN {X -3.1626,Y -112.6066,Z 119,A -94.936,B 24.9529,C -1.5854,E1 24.997,E2 180.8199} C_DIS
LIN {X 0.7947,Y -112.634,Z 119,A -93.4641,B 24.9542,C -1.5626,E1 25.001,E2 179.4018} C_DIS
Enddeposition()
LIN {X 0.7947,Y -112.634,Z 119,A -93.4641,B 24.9542,C -1.5626,E1 25.001,E2 179.4018} C_DIS
Startdeposition()
$VEL.CP = VEL_PRINT
LIN {X -0.4514,Y -111.7584,Z 119,A -94.2931,B 24.9538,C -1.5698,E1 24.9987,E2 180.2138} C_DIS
LIN {X -2.7919,Y -111.726,Z 119,A -95.4923,B 24.9538,C -1.5696,E1 24.9954,E2 181.4136} C_DIS
LIN {X -5.8749,Y -111.6049,Z 119,A -97.0955,B 24.9538,C -1.5686,E1 24.9909,E2 183.0196} C_DIS
LIN {X -8.8792,Y -111.4057,Z 119,A -98.5573,B 24.9537,C -1.5721,E1 24.9868,E2 184.4738} C_DIS
LIN {X -12.3584,Y -111.0755,Z 119,A -100.4117,B 24.9538,C -1.5696,E1 24.9817,E2 186.3351} C_DIS
LIN {X -15.0639,Y -110.7411,Z 119,A -101.9452,B 24.9542,C -1.5641,E1 24.9774,E2 187.8826} C_DIS
LIN {X -18.1269,Y -110.2796,Z 119,A -103.3253,B 24.9536,C -1.5733,E1 24.9736,E2 189.2422} C_DIS
LIN {X -20.8143,Y -109.8041,Z 119,A -104.6401,B 24.9534,C -1.5773,E1 24.97,E2 190.5488} C_DIS
LIN {X -23.5147,Y -109.2576,Z 119,A -106.2159,B 24.9538,C -1.5711,E1 24.9657,E2 192.1412} C_DIS
LIN {X -25.8351,Y -108.734,Z 119,A -107.5716,B 24.9541,C -1.566,E1 24.962,E2 193.5107} C_DIS
LIN {X -28.8467,Y -107.9724,Z 119,A -109.0317,B 24.9537,C -1.5725,E1 24.958,E2 194.9577} C_DIS
LIN {X -31.1277,Y -107.3388,Z 119,A -110.3833,B 24.954,C -1.5676,E1 24.9544,E2 196.3231} C_DIS
LIN {X -34.1004,Y -106.43,Z 119,A -111.9174,B 24.9537,C -1.5713,E1 24.9503,E2 197.8511} C_DIS
LIN {X -37.0566,Y -105.4367,Z 119,A -113.3717,B 24.9533,C -1.5786,E1 24.9465,E2 199.2909} C_DIS
LIN {X -40.6847,Y -104.0907,Z 119,A -115.3988,B 24.9533,C -1.5786,E1 24.9412,E2 201.322} C_DIS
LIN {X -44.3803,Y -102.5698,Z 119,A -117.4641,B 24.9533,C -1.5801,E1 24.9359,E2 203.3886} C_DIS
LIN {X -46.8766,Y -101.4533,Z 119,A -118.8916,B 24.9532,C -1.5806,E1 24.9322,E2 204.8183} C_DIS
LIN {X -49.4621,Y -100.2178,Z 119,A -120.3293,B 24.953,C -1.5837,E1 24.9286,E2 206.2524} C_DIS
LIN {X -51.8045,Y -99.0276,Z 119,A -121.7163,B 24.953,C -1.5837,E1 24.9252,E2 207.6429} C_DIS
LIN {X -54.2198,Y -97.7261,Z 119,A -123.1422,B 24.953,C -1.5849,E1 24.9217,E2 209.0703} C_DIS
LIN {X -56.6297,Y -96.3495,Z 119,A -124.3831,B 24.9524,C -1.5943,E1 24.9187,E2 210.2924} C_DIS
LIN {X -58.9695,Y -94.9355,Z 119,A -125.9537,B 24.9527,C -1.5896,E1 24.9149,E2 211.8792} C_DIS
LIN {X -61.2559,Y -93.4767,Z 119,A -127.1824,B 24.9521,C -1.5983,E1 24.9121,E2 213.0911} C_DIS
LIN {X -63.2137,Y -92.1659,Z 119,A -128.7057,B 24.9528,C -1.5875,E1 24.9085,E2 214.6451} C_DIS
LIN {X -65.469,Y -90.5779,Z 119,A -130.178,B 24.9528,C -1.5875,E1 24.9052,E2 216.1224} C_DIS
LIN {X -68.2853,Y -88.4715,Z 119,A -131.8642,B 24.9523,C -1.5955,E1 24.9014,E2 217.7959} C_DIS
LIN {X -71.0514,Y -86.2671,Z 119,A -133.72,B 24.9523,C -1.5972,E1 24.8974,E2 219.6546} C_DIS
LIN {X -73.518,Y -84.1735,Z 119,A -135.3217,B 24.9519,C -1.6027,E1 24.894,E2 221.2494} C_DIS
LIN {X -76.0615,Y -81.8852,Z 119,A -137.2158,B 24.9519,C -1.6007,E1 24.8901,E2 223.1561} C_DIS
LIN {X -78.5321,Y -79.516,Z 119,A -138.8468,B 24.9515,C -1.6093,E1 24.8869,E2 224.7733} C_DIS
LIN {X -81.2748,Y -76.7107,Z 119,A -140.8853,B 24.9513,C -1.6126,E1 24.8829,E2 226.8126} C_DIS
LIN {X -83.3959,Y -74.3992,Z 119,A -142.5091,B 24.9511,C -1.6157,E1 24.8799,E2 228.4365} C_DIS
LIN {X -85.8361,Y -71.5701,Z 119,A -144.4191,B 24.9508,C -1.6203,E1 24.8764,E2 230.3441} C_DIS
LIN {X -87.7929,Y -69.1557,Z 119,A -146.0356,B 24.9506,C -1.6232,E1 24.8736,E2 231.9612} C_DIS
LIN {X -90.0171,Y -66.235,Z 119,A -147.6671,B 24.9497,C -1.6377,E1 24.8709,E2 233.566} C_DIS
LIN {X -91.6677,Y -63.9308,Z 119,A -149.2933,B 24.9499,C -1.6346,E1 24.8682,E2 235.2077} C_DIS
LIN {X -93.9971,Y -60.4535,Z 119,A -151.4211,B 24.9495,C -1.6408,E1 24.865,E2 237.3312} C_DIS
LIN {X -95.3449,Y -58.3055,Z 119,A -152.6153,B 24.9491,C -1.6484,E1 24.8632,E2 238.5135} C_DIS
LIN {X -96.556,Y -56.2804,Z 119,A -154.0082,B 24.9493,C -1.6445,E1 24.8612,E2 239.923} C_DIS
LIN {X -97.9759,Y -53.7689,Z 119,A -155.4334,B 24.9489,C -1.6506,E1 24.8593,E2 241.341} C_DIS
LIN {X -99.2038,Y -51.4698,Z 119,A -156.977,B 24.9492,C -1.6462,E1 24.8572,E2 242.9033} C_DIS
LIN {X -100.5659,Y -48.7517,Z 119,A -158.4549,B 24.9487,C -1.6538,E1 24.8554,E2 244.3712} C_DIS
LIN {X -101.7667,Y -46.192,Z 119,A -159.6934,B 24.948,C -1.6661,E1 24.854,E2 245.587} C_DIS
LIN {X -102.867,Y -43.6869,Z 119,A -161.1039,B 24.9477,C -1.6699,E1 24.8524,E2 246.9963} C_DIS
LIN {X -103.9058,Y -41.1554,Z 119,A -162.6992,B 24.948,C -1.6665,E1 24.8507,E2 248.6086} C_DIS
LIN {X -104.7639,Y -38.9237,Z 119,A -164.0563,B 24.948,C -1.665,E1 24.8494,E2 249.9768} C_DIS
LIN {X -105.7995,Y -36.0088,Z 119,A -165.3481,B 24.947,C -1.6812,E1 24.8482,E2 251.2374} C_DIS
LIN {X -106.5366,Y -33.7708,Z 119,A -166.8727,B 24.9476,C -1.6726,E1 24.8469,E2 252.7913} C_DIS
LIN {X -107.7149,Y -29.7998,Z 119,A -168.8728,B 24.9469,C -1.6838,E1 24.8454,E2 254.7762} C_DIS
LIN {X -108.5003,Y -26.7929,Z 119,A -170.303,B 24.9462,C -1.6951,E1 24.8444,E2 256.1879} C_DIS
LIN {X -109.0451,Y -24.4891,Z 119,A -171.8355,B 24.9467,C -1.6865,E1 24.8434,E2 257.7498} C_DIS
LIN {X -109.7,Y -21.355,Z 119,A -173.3929,B 24.9462,C -1.695,E1 24.8426,E2 259.2963} C_DIS
LIN {X -110.3435,Y -17.7441,Z 119,A -175.3809,B 24.946,C -1.6968,E1 24.8416,E2 261.2918} C_DIS
LIN {X -110.7923,Y -14.6709,Z 119,A -176.8481,B 24.9454,C -1.7067,E1 24.8411,E2 262.7442} C_DIS
LIN {X -111.1183,Y -11.9546,Z 119,A -178.1564,B 24.9449,C -1.7148,E1 24.8406,E2 264.0409} C_DIS
LIN {X -111.3801,Y -9.2003,Z 119,A -179.6886,B 24.9449,C -1.715,E1 24.8403,E2 265.5819} C_DIS
LIN {X -111.5514,Y -6.8418,Z 119,A 178.9546,B 24.9449,C -1.7133,E1 24.84,E2 266.9508} C_DIS
LIN {X -111.6969,Y -3.7401,Z 119,A 177.6615,B 24.9439,C -1.7299,E1 24.8399,E2 268.212} C_DIS
LIN {X -111.7526,Y -1.3753,Z 119,A 176.1458,B 24.9444,C -1.7222,E1 24.8398,E2 269.7553} C_DIS
LIN {X -111.7461,Y 1.7297,Z 119,A 174.8219,B 24.9434,C -1.7377,E1 24.8398,E2 271.0502} C_DIS
LIN {X -111.685,Y 4.1231,Z 119,A 173.2904,B 24.9439,C -1.73,E1 24.84,E2 272.6093} C_DIS
LIN {X -111.534,Y 7.1024,Z 119,A 172.0027,B 24.943,C -1.7442,E1 24.8401,E2 273.8708} C_DIS
LIN {X -111.3153,Y 9.9545,Z 119,A 170.5811,B 24.9426,C -1.7507,E1 24.8405,E2 275.2854} C_DIS
LIN {X -111.0811,Y 12.3095,Z 119,A 169.1858,B 24.9428,C -1.7477,E1 24.8409,E2 276.6963} C_DIS
LIN {X -110.7445,Y 15.0398,Z 119,A 167.6267,B 24.9428,C -1.7466,E1 24.8414,E2 278.2675} C_DIS
LIN {X -110.2799,Y 18.1252,Z 119,A 166.33,B 24.9417,C -1.7634,E1 24.842,E2 279.5318} C_DIS
LIN {X -109.8029,Y 20.8208,Z 119,A 164.9162,B 24.9414,C -1.7675,E1 24.8427,E2 280.9441} C_DIS
LIN {X -109.26,Y 23.5039,Z 119,A 163.3297,B 24.9416,C -1.765,E1 24.8436,E2 282.546} C_DIS
LIN {X -108.7392,Y 25.8131,Z 119,A 161.9734,B 24.9417,C -1.7634,E1 24.8445,E2 283.914} C_DIS
LIN {X -107.973,Y 28.8446,Z 119,A 160.4052,B 24.9413,C -1.7699,E1 24.8456,E2 285.4759} C_DIS
LIN {X -107.0525,Y 32.0928,Z 119,A 158.5693,B 24.9412,C -1.7714,E1 24.847,E2 287.3189} C_DIS
LIN {X -106.1143,Y 35.0754,Z 119,A 157.1382,B 24.9404,C -1.783,E1 24.8482,E2 288.7305} C_DIS
LIN {X -105.0983,Y 38.007,Z 119,A 155.7093,B 24.9397,C -1.7942,E1 24.8495,E2 290.1408} C_DIS
LIN {X -104.218,Y 40.3605,Z 119,A 154.159,B 24.9401,C -1.7881,E1 24.8511,E2 291.7143} C_DIS
LIN {X -103.2575,Y 42.7601,Z 119,A 152.7707,B 24.94,C -1.7897,E1 24.8525,E2 293.1064} C_DIS
LIN {X -102.181,Y 45.2721,Z 119,A 151.3558,B 24.9397,C -1.7935,E1 24.8541,E2 294.5202} C_DIS
LIN {X -100.8724,Y 48.1137,Z 119,A 150.0485,B 24.9386,C -1.8098,E1 24.8556,E2 295.7957} C_DIS
LIN {X -99.6401,Y 50.6163,Z 119,A 148.4322,B 24.9388,C -1.8069,E1 24.8577,E2 297.4277} C_DIS
LIN {X -98.368,Y 53.046,Z 119,A 147.0299,B 24.9385,C -1.8112,E1 24.8595,E2 298.8271} C_DIS
LIN {X -97.0543,Y 55.4133,Z 119,A 145.6234,B 24.9383,C -1.8145,E1 24.8614,E2 300.233} C_DIS
LIN {X -95.8541,Y 57.4675,Z 119,A 144.4017,B 24.9381,C -1.818,E1 24.8632,E2 301.4529} C_DIS
LIN {X -94.2195,Y 60.1071,Z 119,A 142.7993,B 24.9378,C -1.8221,E1 24.8655,E2 303.0535} C_DIS
LIN {X -92.9278,Y 62.0884,Z 119,A 141.578,B 24.9376,C -1.8252,E1 24.8674,E2 304.2737} C_DIS
LIN {X -91.1186,Y 64.7113,Z 119,A 140.1048,B 24.9368,C -1.836,E1 24.8697,E2 305.7284} C_DIS
LIN {X -89.5213,Y 66.9036,Z 119,A 138.4557,B 24.9372,C -1.8297,E1 24.8725,E2 307.4004} C_DIS
LIN {X -87.6749,Y 69.3051,Z 119,A 136.9262,B 24.9369,C -1.8348,E1 24.8751,E2 308.9249} C_DIS
LIN {X -85.5243,Y 71.9453,Z 119,A 135.1975,B 24.9365,C -1.84,E1 24.8782,E2 310.6492} C_DIS
LIN {X -83.4152,Y 74.3776,Z 119,A 133.4606,B 24.9365,C -1.841,E1 24.8814,E2 312.3917} C_DIS
LIN {X -80.8718,Y 77.1373,Z 119,A 131.4796,B 24.9363,C -1.8436,E1 24.8852,E2 314.3753} C_DIS
LIN {X -78.4601,Y 79.5871,Z 119,A 129.7836,B 24.9358,C -1.8505,E1 24.8885,E2 316.062} C_DIS
LIN {X -75.8,Y 82.1252,Z 119,A 127.8845,B 24.9355,C -1.8544,E1 24.8924,E2 317.9595} C_DIS
LIN {X -73.4652,Y 84.2196,Z 119,A 126.3095,B 24.9352,C -1.8594,E1 24.8957,E2 319.529} C_DIS
LIN {X -70.7389,Y 86.5235,Z 119,A 124.5087,B 24.9348,C -1.8646,E1 24.8995,E2 321.3243} C_DIS
LIN {X -68.3361,Y 88.4323,Z 119,A 123.137,B 24.934,C -1.8759,E1 24.9025,E2 322.6739} C_DIS
LIN {X -66.2466,Y 90.0086,Z 119,A 121.7444,B 24.934,C -1.8767,E1 24.9056,E2 324.0697} C_DIS
LIN {X -64.0295,Y 91.5991,Z 119,A 120.1702,B 24.9343,C -1.8727,E1 24.9092,E2 325.6589} C_DIS
LIN {X -61.7431,Y 93.1555,Z 119,A 118.9349,B 24.9336,C -1.8827,E1 24.912,E2 326.8745} C_DIS
LIN {X -59.3492,Y 94.6983,Z 119,A 117.3295,B 24.9338,C -1.8797,E1 24.9158,E2 328.4921} C_DIS
LIN {X -56.2899,Y 96.5504,Z 119,A 115.3938,B 24.9338,C -1.879,E1 24.9205,E2 330.4354} C_DIS
LIN {X -53.8276,Y 97.9441,Z 119,A 114.0098,B 24.9334,C -1.8842,E1 24.9238,E2 331.811} C_DIS
LIN {X -51.465,Y 99.2063,Z 119,A 112.4676,B 24.9338,C -1.8798,E1 24.9277,E2 333.368} C_DIS
LIN {X -48.76,Y 100.5619,Z 119,A 111.1734,B 24.9329,C -1.8926,E1 24.9309,E2 334.6353} C_DIS
LIN {X -46.1663,Y 101.7783,Z 119,A 109.719,B 24.9327,C -1.8954,E1 24.9345,E2 336.0865} C_DIS
LIN {X -43.642,Y 102.8859,Z 119,A 108.3259,B 24.9324,C -1.8983,E1 24.9381,E2 337.476} C_DIS
LIN {X -41.1286,Y 103.9163,Z 119,A 106.7618,B 24.9328,C -1.8934,E1 24.9422,E2 339.0554} C_DIS
LIN {X -38.9326,Y 104.7607,Z 119,A 105.4162,B 24.9331,C -1.8893,E1 24.9457,E2 340.4133} C_DIS
LIN {X -36.0215,Y 105.7953,Z 119,A 104.117,B 24.9321,C -1.9028,E1 24.9491,E2 341.683} C_DIS
LIN {X -33.7421,Y 106.5458,Z 119,A 102.5922,B 24.9329,C -1.8924,E1 24.9532,E2 343.2354} C_DIS
LIN {X -31.1225,Y 107.3402,Z 119,A 101.3212,B 24.9324,C -1.8992,E1 24.9566,E2 344.4921} C_DIS
LIN {X -28.2059,Y 108.1419,Z 119,A 99.7269,B 24.9324,C -1.8992,E1 24.9609,E2 346.0892} C_DIS
LIN {X -25.7984,Y 108.7426,Z 119,A 98.4932,B 24.9322,C -1.9018,E1 24.9642,E2 347.3181} C_DIS
LIN {X -22.7692,Y 109.4154,Z 119,A 97.0698,B 24.9316,C -1.9101,E1 24.968,E2 348.7237} C_DIS
LIN {X -20.0857,Y 109.9397,Z 119,A 95.6672,B 24.9316,C -1.9112,E1 24.9719,E2 350.1252} C_DIS
LIN {X -17.7554,Y 110.3417,Z 119,A 94.1378,B 24.9324,C -1.8991,E1 24.9762,E2 351.6848} C_DIS
LIN {X -14.6633,Y 110.7933,Z 119,A 92.5913,B 24.9322,C -1.9024,E1 24.9804,E2 353.2247} C_DIS
LIN {X -10.9346,Y 111.2248,Z 119,A 90.6151,B 24.9322,C -1.9013,E1 24.9859,E2 355.2047} C_DIS
LIN {X -7.8434,Y 111.4839,Z 119,A 89.3298,B 24.9313,C -1.9146,E1 24.9894,E2 356.4591} C_DIS
LIN {X -4.9342,Y 111.6501,Z 119,A 87.6992,B 24.9316,C -1.9095,E1 24.994,E2 358.1021} C_DIS
LIN {X -1.3357,Y 111.7529,Z 119,A 85.684,B 24.9321,C -1.903,E1 24.9997,E2 360.133} C_DIS
LIN {X 1.7606,Y 111.7455,Z 119,A 84.1405,B 24.932,C -1.905,E1 25.004,E2 361.6714} C_DIS
LIN {X 5.1147,Y 111.6424,Z 119,A 82.4487,B 24.9319,C -1.9064,E1 25.0087,E2 363.3596} C_DIS
LIN {X 8.2588,Y 111.4553,Z 119,A 80.7604,B 24.9321,C -1.9032,E1 25.0134,E2 365.0546} C_DIS
LIN {X 10.9777,Y 111.2205,Z 119,A 79.4945,B 24.9317,C -1.9086,E1 25.0169,E2 366.307} C_DIS
LIN {X 13.6921,Y 110.9192,Z 119,A 78.0946,B 24.9317,C -1.9084,E1 25.0208,E2 367.7064} C_DIS
LIN {X 16.7642,Y 110.495,Z 119,A 76.4208,B 24.932,C -1.9045,E1 25.0254,E2 369.388} C_DIS
LIN {X 20.8251,Y 109.802,Z 119,A 74.3912,B 24.9318,C -1.9071,E1 25.031,E2 371.409} C_DIS
LIN {X 23.5182,Y 109.2569,Z 119,A 72.9861,B 24.9318,C -1.9066,E1 25.0348,E2 372.8137} C_DIS
LIN {X 25.828,Y 108.7357,Z 119,A 71.6382,B 24.9323,C -1.9003,E1 25.0385,E2 374.1746} C_DIS
LIN {X 28.841,Y 107.974,Z 119,A 70.1826,B 24.932,C -1.9051,E1 25.0424,E2 375.6166} C_DIS
LIN {X 31.685,Y 107.1734,Z 119,A 68.6225,B 24.9322,C -1.9021,E1 25.0466,E2 377.1811} C_DIS
LIN {X 35.1867,Y 106.0767,Z 119,A 66.8166,B 24.9321,C -1.9038,E1 25.0514,E2 378.9797} C_DIS
LIN {X 38.0195,Y 105.0937,Z 119,A 65.4278,B 24.9317,C -1.9087,E1 25.055,E2 380.354} C_DIS
LIN {X 40.2349,Y 104.2674,Z 119,A 63.9143,B 24.9327,C -1.8947,E1 25.059,E2 381.8974} C_DIS
LIN {X 42.7836,Y 103.2477,Z 119,A 62.5138,B 24.9327,C -1.8935,E1 25.0627,E2 383.2976} C_DIS
LIN {X 45.2858,Y 102.175,Z 119,A 61.1112,B 24.9329,C -1.8916,E1 25.0663,E2 384.7012} C_DIS
LIN {X 48.127,Y 100.8661,Z 119,A 59.8233,B 24.9321,C -1.9033,E1 25.0694,E2 385.9582} C_DIS
LIN {X 50.5836,Y 99.6568,Z 119,A 58.2027,B 24.9329,C -1.8922,E1 25.0735,E2 387.6007} C_DIS
LIN {X 53.1117,Y 98.3324,Z 119,A 56.8026,B 24.9329,C -1.8929,E1 25.077,E2 388.9951} C_DIS
LIN {X 55.4568,Y 97.0293,Z 119,A 55.428,B 24.9329,C -1.891,E1 25.0803,E2 390.3701} C_DIS
LIN {X 57.5041,Y 95.8319,Z 119,A 54.1144,B 24.9334,C -1.8849,E1 25.0835,E2 391.6941} C_DIS
LIN {X 60.1105,Y 94.2173,Z 119,A 52.6433,B 24.9333,C -1.8869,E1 25.087,E2 393.1558} C_DIS
LIN {X 62.093,Y 92.9247,Z 119,A 51.4342,B 24.9333,C -1.885,E1 25.0898,E2 394.3653} C_DIS
LIN {X 64.6583,Y 91.1564,Z 119,A 49.8115,B 24.9337,C -1.8813,E1 25.0935,E2 395.9914} C_DIS
LIN {X 67.1286,Y 89.3523,Z 119,A 48.2399,B 24.9339,C -1.8783,E1 25.097,E2 397.5643} C_DIS
LIN {X 69.8438,Y 87.2489,Z 119,A 46.4521,B 24.9342,C -1.8739,E1 25.101,E2 399.3559} C_DIS
LIN {X 72.3483,Y 85.1812,Z 119,A 44.8244,B 24.9342,C -1.8723,E1 25.1044,E2 400.9811} C_DIS
LIN {X 74.6757,Y 83.1483,Z 119,A 43.1937,B 24.9347,C -1.8671,E1 25.1079,E2 402.6177} C_DIS
LIN {X 77.4254,Y 80.5942,Z 119,A 41.3147,B 24.9347,C -1.8651,E1 25.1117,E2 404.4937} C_DIS
LIN {X 79.655,Y 78.3914,Z 119,A 39.7096,B 24.935,C -1.8617,E1 25.1148,E2 406.1} C_DIS
LIN {X 82.0156,Y 75.9194,Z 119,A 37.9308,B 24.9354,C -1.8566,E1 25.1183,E2 407.883} C_DIS
LIN {X 84.1759,Y 73.5153,Z 119,A 36.3449,B 24.9354,C -1.8559,E1 25.1212,E2 409.4635} C_DIS
LIN {X 86.3853,Y 70.9092,Z 119,A 34.5617,B 24.9358,C -1.8504,E1 25.1244,E2 411.2516} C_DIS
LIN {X 88.9436,Y 67.6726,Z 119,A 32.3877,B 24.9364,C -1.8426,E1 25.1281,E2 413.4336} C_DIS
LIN {X 90.5814,Y 65.4641,Z 119,A 30.9996,B 24.9365,C -1.84,E1 25.1304,E2 414.8212} C_DIS
LIN {X 92.3641,Y 62.921,Z 119,A 29.7209,B 24.9359,C -1.8499,E1 25.1324,E2 416.0703} C_DIS
LIN {X 93.6766,Y 60.9527,Z 119,A 28.2117,B 24.937,C -1.8335,E1 25.1348,E2 417.6106} C_DIS
LIN {X 95.3475,Y 58.3011,Z 119,A 26.917,B 24.9363,C -1.8432,E1 25.1366,E2 418.8759} C_DIS
LIN {X 96.5623,Y 56.2695,Z 119,A 25.5406,B 24.937,C -1.8326,E1 25.1386,E2 420.2702} C_DIS
LIN {X 97.9116,Y 53.8875,Z 119,A 24.145,B 24.9373,C -1.8291,E1 25.1405,E2 421.6667} C_DIS
LIN {X 99.2622,Y 51.3557,Z 119,A 22.5836,B 24.9378,C -1.821,E1 25.1426,E2 423.2392} C_DIS
LIN {X 100.4509,Y 48.9911,Z 119,A 21.337,B 24.9378,C -1.8221,E1 25.1441,E2 424.4765} C_DIS
LIN {X 101.7678,Y 46.1896,Z 119,A 19.9286,B 24.9375,C -1.8256,E1 25.1457,E2 425.869} C_DIS
LIN {X 102.865,Y 43.6917,Z 119,A 18.5373,B 24.9378,C -1.8218,E1 25.1473,E2 427.2615} C_DIS
LIN {X 103.9009,Y 41.1679,Z 119,A 16.9699,B 24.9386,C -1.8101,E1 25.1489,E2 428.8478} C_DIS
LIN {X 104.9579,Y 38.3917,Z 119,A 15.5291,B 24.9386,C -1.8093,E1 25.1503,E2 430.2826} C_DIS
LIN {X 105.8003,Y 36.0067,Z 119,A 14.3453,B 24.9386,C -1.8105,E1 25.1514,E2 431.4569} C_DIS
LIN {X 106.6017,Y 33.5618,Z 119,A 12.7587,B 24.9396,C -1.7944,E1 25.1528,E2 433.0724} C_DIS
LIN {X 107.7143,Y 29.8022,Z 119,A 10.8684,B 24.9397,C -1.7936,E1 25.1543,E2 434.9538} C_DIS
LIN {X 108.4995,Y 26.7963,Z 119,A 9.456,B 24.9395,C -1.7969,E1 25.1552,E2 436.3504} C_DIS
LIN {X 109.0482,Y 24.475,Z 119,A 7.9379,B 24.9406,C -1.7797,E1 25.1562,E2 437.9002} C_DIS
LIN {X 109.7177,Y 21.2629,Z 119,A 6.4402,B 24.9404,C -1.7828,E1 25.157,E2 439.3819} C_DIS
LIN {X 110.3453,Y 17.7321,Z 119,A 4.4444,B 24.9413,C -1.7698,E1 25.158,E2 441.3967} C_DIS
LIN {X 110.7915,Y 14.6776,Z 119,A 2.9271,B 24.9414,C -1.7677,E1 25.1586,E2 442.9099} C_DIS
LIN {X 111.2346,Y 10.8287,Z 119,A 0.9169,B 24.9419,C -1.7602,E1 25.1592,E2 444.9258} C_DIS
LIN {X 111.4873,Y 7.7932,Z 119,A -0.3506,B 24.9414,C -1.7685,E1 25.1594,E2 446.1662} C_DIS
LIN {X 111.6432,Y 5.0958,Z 119,A -1.8917,B 24.9421,C -1.757,E1 25.1597,E2 447.7255} C_DIS
LIN {X 111.7291,Y 2.6527,Z 119,A -3.1318,B 24.9424,C -1.7535,E1 25.1597,E2 448.9664} C_DIS
LIN {X 111.7589,Y -0.3413,Z 119,A -4.6854,B 24.9428,C -1.7477,E1 25.1597,E2 450.5244} C_DIS
LIN {X 111.7265,Y -2.7752,Z 119,A -5.9013,B 24.9429,C -1.745,E1 25.1597,E2 451.7394} C_DIS
LIN {X 111.6054,Y -5.8651,Z 119,A -7.439,B 24.9431,C -1.742,E1 25.1595,E2 453.275} C_DIS
LIN {X 111.4586,Y -8.2172,Z 119,A -8.8225,B 24.9439,C -1.7301,E1 25.1593,E2 454.6784} C_DIS
LIN {X 111.221,Y -10.9731,Z 119,A -10.0843,B 24.9437,C -1.7326,E1 25.1589,E2 455.9269} C_DIS
LIN {X 110.9204,Y -13.6825,Z 119,A -11.4874,B 24.9441,C -1.7277,E1 25.1585,E2 457.333} C_DIS
LIN {X 110.4921,Y -16.7827,Z 119,A -13.0671,B 24.9443,C -1.7237,E1 25.1578,E2 458.913} C_DIS
LIN {X 110.0587,Y -19.4239,Z 119,A -14.448,B 24.9446,C -1.7188,E1 25.1572,E2 460.2973} C_DIS
LIN {X 109.615,Y -21.7965,Z 119,A -15.8008,B 24.9452,C -1.7096,E1 25.1565,E2 461.664} C_DIS
LIN {X 108.959,Y -24.8617,Z 119,A -17.0862,B 24.9446,C -1.719,E1 25.1557,E2 462.9197} C_DIS
LIN {X 108.3174,Y -27.5228,Z 119,A -18.6497,B 24.9454,C -1.7072,E1 25.1547,E2 464.5019} C_DIS
LIN {X 107.3386,Y -31.1284,Z 119,A -20.687,B 24.9461,C -1.6955,E1 25.1531,E2 466.5551} C_DIS
LIN {X 106.43,Y -34.1004,Z 119,A -21.9663,B 24.9455,C -1.7048,E1 25.1521,E2 467.8053} C_DIS
LIN {X 105.6854,Y -36.3475,Z 119,A -23.4723,B 24.9466,C -1.6876,E1 25.1507,E2 469.3433} C_DIS
LIN {X 104.7636,Y -38.9246,Z 119,A -24.8046,B 24.9467,C -1.6864,E1 25.1494,E2 470.6709} C_DIS
LIN {X 103.6197,Y -41.8703,Z 119,A -26.1731,B 24.9463,C -1.6928,E1 25.1481,E2 472.0168} C_DIS
LIN {X 102.568,Y -44.3843,Z 119,A -27.5584,B 24.9465,C -1.6891,E1 25.1466,E2 473.4033} C_DIS
LIN {X 101.4549,Y -46.8731,Z 119,A -29.1256,B 24.9473,C -1.6771,E1 25.1447,E2 474.9903} C_DIS
LIN {X 100.4331,Y -49.0278,Z 119,A -30.4681,B 24.9479,C -1.6679,E1 25.1431,E2 476.3472} C_DIS
LIN {X 99.0307,Y -51.7987,Z 119,A -31.9158,B 24.9478,C -1.6697,E1 25.1412,E2 477.783} C_DIS
LIN {X 97.7332,Y -54.2071,Z 119,A -33.3887,B 24.9482,C -1.6624,E1 25.1392,E2 479.2655} C_DIS
LIN {X 95.7977,Y -57.5604,Z 119,A -35.2653,B 24.9482,C -1.6614,E1 25.1366,E2 481.1346} C_DIS
LIN {X 94.1996,Y -60.1381,Z 119,A -36.8193,B 24.9485,C -1.657,E1 25.1343,E2 482.6912} C_DIS
LIN {X 92.8586,Y -62.1906,Z 119,A -38.2054,B 24.9491,C -1.6476,E1 25.1321,E2 484.0926} C_DIS
LIN {X 90.5728,Y -65.4759,Z 119,A -40.2509,B 24.9495,C -1.6422,E1 25.1288,E2 486.141} C_DIS
LIN {X 88.5244,Y -68.2166,Z 119,A -41.861,B 24.9494,C -1.6439,E1 25.1261,E2 487.7393} C_DIS
LIN {X 86.8263,Y -70.3653,Z 119,A -43.3071,B 24.9497,C -1.6382,E1 25.1236,E2 489.192} C_DIS
LIN {X 84.4994,Y -73.1449,Z 119,A -45.2064,B 24.9501,C -1.6315,E1 25.1202,E2 491.0986} C_DIS
LIN {X 82.3449,Y -75.5605,Z 119,A -46.7553,B 24.9501,C -1.6322,E1 25.1173,E2 492.6389} C_DIS
LIN {X 80.3403,Y -77.6888,Z 119,A -48.3086,B 24.9505,C -1.626,E1 25.1143,E2 494.2002} C_DIS
LIN {X 77.6845,Y -80.3444,Z 119,A -50.2087,B 24.9507,C -1.6224,E1 25.1105,E2 496.1007} C_DIS
LIN {X 75.5555,Y -82.3495,Z 119,A -51.691,B 24.9508,C -1.6196,E1 25.1074,E2 497.5836} C_DIS
LIN {X 72.9993,Y -84.6265,Z 119,A -53.5692,B 24.9514,C -1.61,E1 25.1035,E2 499.4771} C_DIS
LIN {X 70.3719,Y -86.821,Z 119,A -55.2055,B 24.9514,C -1.6114,E1 25.1,E2 501.1038} C_DIS
LIN {X 67.5127,Y -89.0637,Z 119,A -57.0637,B 24.9516,C -1.6075,E1 25.0959,E2 502.9643} C_DIS
LIN {X 65.4651,Y -90.5807,Z 119,A -58.435,B 24.9519,C -1.6019,E1 25.0927,E2 504.3441} C_DIS
LIN {X 62.9203,Y -92.3646,Z 119,A -59.7161,B 24.9513,C -1.6125,E1 25.0899,E2 505.5957} C_DIS
LIN {X 60.9506,Y -93.678,Z 119,A -61.3399,B 24.9525,C -1.5919,E1 25.086,E2 507.2628} C_DIS
LIN {X 57.4209,Y -95.8819,Z 119,A -63.218,B 24.9521,C -1.5991,E1 25.0816,E2 509.118} C_DIS
LIN {X 55.0615,Y -97.256,Z 119,A -64.6131,B 24.9522,C -1.5968,E1 25.0782,E2 510.5144} C_DIS
LIN {X 52.6674,Y -98.5731,Z 119,A -66.0089,B 24.9524,C -1.5945,E1 25.0747,E2 511.9115} C_DIS
LIN {X 49.9094,Y -99.9961,Z 119,A -67.4235,B 24.9521,C -1.5997,E1 25.0713,E2 513.3101} C_DIS
LIN {X 47.7835,Y -101.0311,Z 119,A -68.9529,B 24.953,C -1.5837,E1 25.0673,E2 514.8731} C_DIS
LIN {X 45.2579,Y -102.1872,Z 119,A -70.3511,B 24.953,C -1.5827,E1 25.0638,E2 516.2705} C_DIS
LIN {X 42.5455,Y -103.3448,Z 119,A -71.7741,B 24.953,C -1.5843,E1 25.0601,E2 517.6862} C_DIS
LIN {X 39.8933,Y -104.3969,Z 119,A -73.026,B 24.9525,C -1.5915,E1 25.0569,E2 518.9182} C_DIS
LIN {X 37.3018,Y -105.3506,Z 119,A -74.6871,B 24.9533,C -1.5789,E1 25.0525,E2 520.6057} C_DIS
LIN {X 34.3648,Y -106.3444,Z 119,A -76.2384,B 24.9533,C -1.5786,E1 25.0484,E2 522.1547} C_DIS
LIN {X 31.116,Y -107.3421,Z 119,A -77.9229,B 24.9533,C -1.5791,E1 25.0439,E2 523.8352} C_DIS
LIN {X 28.4782,Y -108.0719,Z 119,A -79.4584,B 24.9537,C -1.5719,E1 25.0397,E2 525.3854} C_DIS
LIN {X 25.6478,Y -108.7774,Z 119,A -80.7626,B 24.9533,C -1.5787,E1 25.0362,E2 526.6716} C_DIS
LIN {X 22.74,Y -109.4214,Z 119,A -82.1711,B 24.9531,C -1.5824,E1 25.0324,E2 528.0695} C_DIS
LIN {X 20.0661,Y -109.9432,Z 119,A -83.5628,B 24.9531,C -1.5814,E1 25.0286,E2 529.4619} C_DIS
LIN {X 17.7419,Y -110.3438,Z 119,A -85.0739,B 24.954,C -1.5675,E1 25.0243,E2 531.0044} C_DIS
LIN {X 14.5993,Y -110.8016,Z 119,A -86.5523,B 24.9537,C -1.5728,E1 25.0203,E2 532.4689} C_DIS
LIN {X 11.9317,Y -111.1207,Z 119,A -87.7696,B 24.9533,C -1.5788,E1 25.017,E2 533.671} C_DIS
LIN {X 9.1768,Y -111.3819,Z 119,A -89.357,B 24.9538,C -1.5709,E1 25.0125,E2 535.2764} C_DIS
LIN {X 6.8283,Y -111.5522,Z 119,A -90.6967,B 24.9541,C -1.5647,E1 25.0087,E2 536.6302} C_DIS
LIN {X 3.7367,Y -111.697,Z 119,A -92.1883,B 24.9539,C -1.5681,E1 25.0046,E2 538.1132} C_DIS
LIN {X 0.7922,Y -111.7547,Z 119,A -93.5594,B 24.9536,C -1.5737,E1 25.0008,E2 539.471} C_DIS
Enddeposition()
LIN {X 0.8293,Y -117.7293,Z 120,A -93.0051,B 24.9578,C -1.5008,E1 25.0019,E2 539.0895} C_DIS
Startdeposition()
$VEL.CP = VEL_PRINT
LIN {X 4.3335,Y -117.656,Z 120,A -90.9751,B 24.9569,C -1.5161,E1 25.0076,E2 537.0236} C_DIS
LIN {X 7.2196,Y -117.5143,Z 120,A -89.57,B 24.9569,C -1.5166,E1 25.0115,E2 535.6178} C_DIS
LIN {X 10.5027,Y -117.2646,Z 120,A -88.2845,B 24.9577,C -1.5029,E1 25.015,E2 534.3655} C_DIS
LIN {X 12.9771,Y -117.0185,Z 120,A -86.7608,B 24.9568,C -1.518,E1 25.0193,E2 532.8071} C_DIS
LIN {X 16.2439,Y -116.6081,Z 120,A -85.4756,B 24.9576,C -1.5045,E1 25.0228,E2 531.555} C_DIS
LIN {X 19.1007,Y -116.1743,Z 120,A -84.0715,B 24.9576,C -1.5054,E1 25.0267,E2 530.15} C_DIS
LIN {X 21.946,Y -115.6705,Z 120,A -82.6677,B 24.9575,C -1.5064,E1 25.0306,E2 528.7453} C_DIS
LIN {X 24.7781,Y -115.0971,Z 120,A -81.2638,B 24.9575,C -1.5075,E1 25.0344,E2 527.3406} C_DIS
LIN {X 27.5953,Y -114.4544,Z 120,A -79.8607,B 24.9574,C -1.5087,E1 25.0382,E2 525.9365} C_DIS
LIN {X 30.3958,Y -113.7427,Z 120,A -78.2811,B 24.9568,C -1.5182,E1 25.0425,E2 524.3368} C_DIS
LIN {X 33.1937,Y -112.9578,Z 120,A -77.0539,B 24.9572,C -1.5111,E1 25.0458,E2 523.1286} C_DIS
LIN {X 35.9403,Y -112.1142,Z 120,A -75.6522,B 24.9572,C -1.5129,E1 25.0495,E2 521.725} C_DIS
LIN {X 38.3007,Y -111.3319,Z 120,A -74.2685,B 24.9566,C -1.5225,E1 25.0532,E2 520.3214} C_DIS
LIN {X 41.0214,Y -110.3584,Z 120,A -72.8664,B 24.9565,C -1.5242,E1 25.0569,E2 518.9182} C_DIS
LIN {X 43.7173,Y -109.3184,Z 120,A -71.3264,B 24.956,C -1.5325,E1 25.061,E2 517.362} C_DIS
LIN {X 46.387,Y -108.2126,Z 120,A -70.0625,B 24.9563,C -1.5279,E1 25.0642,E2 516.1121} C_DIS
LIN {X 49.0287,Y -107.0416,Z 120,A -68.661,B 24.9562,C -1.5298,E1 25.0677,E2 514.7094} C_DIS
LIN {X 51.6408,Y -105.8062,Z 120,A -67.1217,B 24.9557,C -1.5384,E1 25.0717,E2 513.1539} C_DIS
LIN {X 54.5784,Y -104.3192,Z 120,A -65.8393,B 24.9564,C -1.5261,E1 25.0748,E2 511.9043} C_DIS
LIN {X 57.1221,Y -102.9484,Z 120,A -64.4386,B 24.9562,C -1.5283,E1 25.0782,E2 510.5023} C_DIS
LIN {X 59.2845,Y -101.7206,Z 120,A -62.9188,B 24.9553,C -1.5451,E1 25.082,E2 508.9473} C_DIS
LIN {X 62.1047,Y -100.0215,Z 120,A -61.6371,B 24.956,C -1.533,E1 25.0849,E2 507.6983} C_DIS
LIN {X 64.5407,Y -98.4673,Z 120,A -60.0604,B 24.9553,C -1.5438,E1 25.0887,E2 506.1011} C_DIS
LIN {X 66.9378,Y -96.8537,Z 120,A -58.6604,B 24.9552,C -1.5464,E1 25.0919,E2 504.6998} C_DIS
LIN {X 69.2945,Y -95.1818,Z 120,A -57.2603,B 24.955,C -1.549,E1 25.0951,E2 503.2984} C_DIS
LIN {X 71.6095,Y -93.4526,Z 120,A -55.7933,B 24.9547,C -1.555,E1 25.0984,E2 501.8228} C_DIS
LIN {X 74.2109,Y -91.4,Z 120,A -54.2204,B 24.9546,C -1.5566,E1 25.1018,E2 500.2518} C_DIS
LIN {X 77.2053,Y -88.8855,Z 120,A -52.5379,B 24.955,C -1.5505,E1 25.1054,E2 498.5904} C_DIS
LIN {X 79.0665,Y -87.2365,Z 120,A -51.0052,B 24.9539,C -1.5687,E1 25.1086,E2 497.0207} C_DIS
LIN {X 81.1836,Y -85.2698,Z 120,A -49.7586,B 24.9541,C -1.5644,E1 25.1111,E2 495.7894} C_DIS
LIN {X 83.535,Y -82.9651,Z 120,A -48.1646,B 24.9539,C -1.568,E1 25.1143,E2 494.1937} C_DIS
LIN {X 85.7101,Y -80.7155,Z 120,A -46.7197,B 24.9539,C -1.568,E1 25.117,E2 492.7547} C_DIS
LIN {X 87.5053,Y -78.7663,Z 120,A -45.5435,B 24.9541,C -1.566,E1 25.1192,E2 491.5888} C_DIS
LIN {X 89.1506,Y -76.9018,Z 120,A -44.0262,B 24.953,C -1.5839,E1 25.1221,E2 490.0361} C_DIS
LIN {X 91.2647,Y -74.3778,Z 120,A -42.5706,B 24.9532,C -1.5811,E1 25.1247,E2 488.5938} C_DIS
LIN {X 92.8941,Y -72.3343,Z 120,A -41.3616,B 24.9532,C -1.5815,E1 25.1267,E2 487.3895} C_DIS
LIN {X 94.5663,Y -70.1351,Z 120,A -39.9692,B 24.9528,C -1.5875,E1 25.1291,E2 485.9897} C_DIS
LIN {X 96.259,Y -67.7933,Z 120,A -38.5713,B 24.9526,C -1.591,E1 25.1313,E2 484.5903} C_DIS
LIN {X 97.8938,Y -65.4105,Z 120,A -37.0362,B 24.952,C -1.6012,E1 25.1338,E2 483.0387} C_DIS
LIN {X 99.4695,Y -62.9884,Z 120,A -35.776,B 24.9521,C -1.5982,E1 25.1356,E2 481.792} C_DIS
LIN {X 101.1904,Y -60.1814,Z 120,A -34.1836,B 24.9519,C -1.6024,E1 25.138,E2 480.1977} C_DIS
LIN {X 102.4404,Y -58.0318,Z 120,A -32.8435,B 24.9513,C -1.6122,E1 25.1398,E2 478.8414} C_DIS
LIN {X 103.8337,Y -55.5003,Z 120,A -31.5837,B 24.9515,C -1.6093,E1 25.1415,E2 477.5951} C_DIS
LIN {X 105.3435,Y -52.5743,Z 120,A -29.9917,B 24.9512,C -1.6136,E1 25.1435,E2 476.0013} C_DIS
LIN {X 106.602,Y -49.9732,Z 120,A -28.5944,B 24.951,C -1.6175,E1 25.1452,E2 474.6025} C_DIS
LIN {X 107.7963,Y -47.342,Z 120,A -27.1557,B 24.9506,C -1.6234,E1 25.1468,E2 473.1577} C_DIS
LIN {X 108.9256,Y -44.6823,Z 120,A -25.8004,B 24.9506,C -1.6253,E1 25.1483,E2 471.8055} C_DIS
LIN {X 109.9894,Y -41.9957,Z 120,A -24.4036,B 24.9503,C -1.6292,E1 25.1497,E2 470.4071} C_DIS
LIN {X 110.9869,Y -39.2838,Z 120,A -23.0067,B 24.95,C -1.6332,E1 25.151,E2 469.0087} C_DIS
LIN {X 111.7935,Y -36.9316,Z 120,A -21.6525,B 24.9494,C -1.644,E1 25.1522,E2 467.6366} C_DIS
LIN {X 112.6662,Y -34.1769,Z 120,A -20.2645,B 24.9491,C -1.6476,E1 25.1534,E2 466.2481} C_DIS
LIN {X 113.506,Y -31.272,Z 120,A -18.8566,B 24.9491,C -1.6492,E1 25.1544,E2 464.8444} C_DIS
LIN {X 114.2074,Y -28.6075,Z 120,A -17.4771,B 24.9487,C -1.6554,E1 25.1554,E2 463.4584} C_DIS
LIN {X 114.8751,Y -25.7961,Z 120,A -16.0806,B 24.9484,C -1.6594,E1 25.1562,E2 462.0603} C_DIS
LIN {X 115.4736,Y -22.9691,Z 120,A -14.6839,B 24.9481,C -1.6635,E1 25.157,E2 460.6622} C_DIS
LIN {X 116.0025,Y -20.1283,Z 120,A -13.2874,B 24.9479,C -1.6676,E1 25.1577,E2 459.2642} C_DIS
LIN {X 116.4615,Y -17.2754,Z 120,A -12.0283,B 24.9481,C -1.665,E1 25.1582,E2 458.0187} C_DIS
LIN {X 116.8973,Y -14.0119,Z 120,A -10.4371,B 24.9478,C -1.6697,E1 25.1588,E2 456.4257} C_DIS
LIN {X 117.1689,Y -11.5401,Z 120,A -9.2353,B 24.9475,C -1.6732,E1 25.1591,E2 455.2227} C_DIS
LIN {X 117.444,Y -8.2592,Z 120,A -7.6067,B 24.9471,C -1.6798,E1 25.1595,E2 453.5884} C_DIS
LIN {X 117.6113,Y -5.3745,Z 120,A -6.2474,B 24.947,C -1.6821,E1 25.1597,E2 452.2317} C_DIS
LIN {X 117.7004,Y -2.8894,Z 120,A -5.0459,B 24.9468,C -1.6856,E1 25.1597,E2 451.0291} C_DIS
LIN {X 117.7356,Y 0,Z 120,A -3.5047,B 24.946,C -1.6968,E1 25.1597,E2 449.4707} C_DIS
LIN {X 117.688,Y 3.2921,Z 120,A -2.2342,B 24.9467,C -1.6859,E1 25.1597,E2 448.2334} C_DIS
LIN {X 117.5718,Y 6.1793,Z 120,A -0.8373,B 24.9465,C -1.69,E1 25.1595,E2 446.8351} C_DIS
LIN {X 117.3847,Y 9.0628,Z 120,A 0.7348,B 24.9457,C -1.7026,E1 25.1592,E2 445.2427} C_DIS
LIN {X 117.1689,Y 11.5401,Z 120,A 1.9369,B 24.9455,C -1.7061,E1 25.1589,E2 444.0396} C_DIS
LIN {X 116.8504,Y 14.4121,Z 120,A 3.4711,B 24.9448,C -1.7168,E1 25.1584,E2 442.489} C_DIS
LIN {X 116.4615,Y 17.2754,Z 120,A 4.8675,B 24.9445,C -1.7208,E1 25.1578,E2 441.0914} C_DIS
LIN {X 116.0025,Y 20.1283,Z 120,A 6.2644,B 24.9442,C -1.7248,E1 25.1572,E2 439.6933} C_DIS
LIN {X 115.4736,Y 22.9691,Z 120,A 7.5237,B 24.9444,C -1.7221,E1 25.1565,E2 438.4477} C_DIS
LIN {X 114.7844,Y 26.1887,Z 120,A 9.1155,B 24.9441,C -1.7267,E1 25.1556,E2 436.8544} C_DIS
LIN {X 114.1933,Y 28.6625,Z 120,A 10.4619,B 24.9435,C -1.7358,E1 25.1547,E2 435.4943} C_DIS
LIN {X 113.3611,Y 31.7893,Z 120,A 11.9092,B 24.9436,C -1.7345,E1 25.1536,E2 434.0583} C_DIS
LIN {X 112.5051,Y 34.6962,Z 120,A 13.3319,B 24.9435,C -1.7365,E1 25.1525,E2 432.639} C_DIS
LIN {X 111.3319,Y 38.3007,Z 120,A 15.2075,B 24.943,C -1.7436,E1 25.1508,E2 430.7574} C_DIS
LIN {X 110.2157,Y 41.3982,Z 120,A 16.6234,B 24.9433,C -1.7394,E1 25.1495,E2 429.3593} C_DIS
LIN {X 109.3184,Y 43.7173,Z 120,A 18.1397,B 24.9421,C -1.7577,E1 25.1479,E2 427.8082} C_DIS
LIN {X 108.2126,Y 46.387,Z 120,A 19.5372,B 24.9419,C -1.7614,E1 25.1463,E2 426.4097} C_DIS
LIN {X 106.8716,Y 49.394,Z 120,A 20.816,B 24.9426,C -1.7505,E1 25.1449,E2 425.1636} C_DIS
LIN {X 105.8062,Y 51.6408,Z 120,A 22.3325,B 24.9414,C -1.7686,E1 25.143,E2 423.6124} C_DIS
LIN {X 104.3192,Y 54.5784,Z 120,A 23.7875,B 24.9415,C -1.766,E1 25.1412,E2 422.1712} C_DIS
LIN {X 102.9484,Y 57.1221,Z 120,A 25.1857,B 24.9413,C -1.7695,E1 25.1393,E2 420.772} C_DIS
LIN {X 101.7206,Y 59.2845,Z 120,A 26.3887,B 24.9411,C -1.7725,E1 25.1376,E2 419.5684} C_DIS
LIN {X 100.0215,Y 62.1047,Z 120,A 28.0257,B 24.9407,C -1.7784,E1 25.1352,E2 417.9256} C_DIS
LIN {X 97.8938,Y 65.4105,Z 120,A 29.8847,B 24.9406,C -1.7808,E1 25.1324,E2 416.0703} C_DIS
LIN {X 96.259,Y 67.7932,Z 120,A 31.283,B 24.9403,C -1.784,E1 25.1302,E2 414.6712} C_DIS
LIN {X 94.5663,Y 70.1351,Z 120,A 32.682,B 24.9401,C -1.7872,E1 25.1278,E2 413.2715} C_DIS
LIN {X 92.5668,Y 72.7509,Z 120,A 34.276,B 24.9399,C -1.7908,E1 25.1251,E2 411.6766} C_DIS
LIN {X 91.011,Y 74.6908,Z 120,A 35.4798,B 24.9397,C -1.7934,E1 25.123,E2 410.4723} C_DIS
LIN {X 89.1506,Y 76.9018,Z 120,A 36.8793,B 24.9395,C -1.7963,E1 25.1205,E2 409.0722} C_DIS
LIN {X 86.9641,Y 79.3634,Z 120,A 38.4737,B 24.9393,C -1.7997,E1 25.1175,E2 407.477} C_DIS
LIN {X 84.9902,Y 81.4737,Z 120,A 39.8732,B 24.9391,C -1.8025,E1 25.1148,E2 406.077} C_DIS
LIN {X 82.2239,Y 84.2672,Z 120,A 41.9155,B 24.9384,C -1.8127,E1 25.1107,E2 404.0192} C_DIS
LIN {X 80.1311,Y 86.2597,Z 120,A 43.3155,B 24.9382,C -1.8153,E1 25.1079,E2 402.6187} C_DIS
LIN {X 77.6866,Y 88.4652,Z 120,A 44.773,B 24.9385,C -1.8117,E1 25.1049,E2 401.1754} C_DIS
LIN {X 75.4921,Y 90.3451,Z 120,A 45.9967,B 24.9389,C -1.8059,E1 25.1023,E2 399.9702} C_DIS
LIN {X 73.2961,Y 92.1359,Z 120,A 47.565,B 24.9381,C -1.8174,E1 25.0988,E2 398.3808} C_DIS
LIN {X 70.9682,Y 93.9405,Z 120,A 48.9748,B 24.938,C -1.8189,E1 25.0957,E2 396.9725} C_DIS
LIN {X 68.9694,Y 95.4198,Z 120,A 50.2333,B 24.9377,C -1.8232,E1 25.0929,E2 395.7082} C_DIS
LIN {X 66.2732,Y 97.3096,Z 120,A 51.777,B 24.9377,C -1.8232,E1 25.0893,E2 394.1698} C_DIS
LIN {X 63.8652,Y 98.9067,Z 120,A 53.1784,B 24.9376,C -1.8253,E1 25.086,E2 392.7681} C_DIS
LIN {X 61.4187,Y 100.4443,Z 120,A 54.58,B 24.9374,C -1.8272,E1 25.0827,E2 391.3663} C_DIS
LIN {X 58.9351,Y 101.9213,Z 120,A 55.9819,B 24.9373,C -1.8291,E1 25.0793,E2 389.9643} C_DIS
LIN {X 56.4161,Y 103.337,Z 120,A 57.3839,B 24.9372,C -1.8309,E1 25.0759,E2 388.5622} C_DIS
LIN {X 53.7966,Y 104.7244,Z 120,A 58.7992,B 24.9372,C -1.8316,E1 25.0724,E2 387.1492} C_DIS
LIN {X 51.2776,Y 105.9807,Z 120,A 60.0118,B 24.9375,C -1.826,E1 25.0694,E2 385.953} C_DIS
LIN {X 48.6613,Y 107.2072,Z 120,A 61.5913,B 24.9368,C -1.8357,E1 25.0654,E2 384.3547} C_DIS
LIN {X 46.387,Y 108.2126,Z 120,A 62.7986,B 24.9368,C -1.8369,E1 25.0623,E2 383.1474} C_DIS
LIN {X 43.7173,Y 109.3184,Z 120,A 64.3673,B 24.9361,C -1.8458,E1 25.0582,E2 381.5612} C_DIS
LIN {X 41.0214,Y 110.3584,Z 120,A 65.7434,B 24.9361,C -1.8458,E1 25.0546,E2 380.1881} C_DIS
LIN {X 37.9188,Y 111.4606,Z 120,A 67.0273,B 24.937,C -1.8326,E1 25.0513,E2 378.9378} C_DIS
LIN {X 35.172,Y 112.3576,Z 120,A 68.6081,B 24.9364,C -1.8417,E1 25.047,E2 377.3385} C_DIS
LIN {X 32.4041,Y 113.1869,Z 120,A 70.0124,B 24.9364,C -1.8427,E1 25.0433,E2 375.9343} C_DIS
Enddeposition()
END
